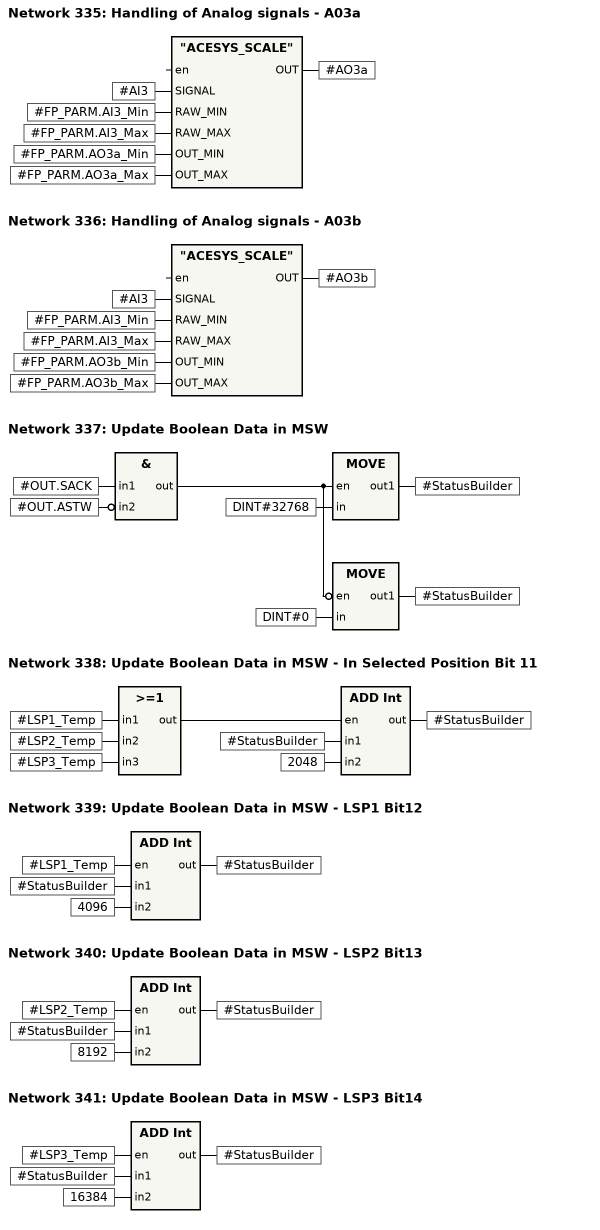
   "ACESYS_SCALE"(SIGNAL := #AI3,
                  RAW_MIN := #FP_PARM.AI3_Min,
                  RAW_MAX := #FP_PARM.AI3_Max,
                  OUT_MIN := #FP_PARM.AO3a_Min,
                  OUT_MAX := #FP_PARM.AO3a_Max,
                  OUT => #AO3a);
END_REGION

REGION Network 336: Handling of Analog signals - A03b
   "ACESYS_SCALE"(SIGNAL := #AI3,
                  RAW_MIN := #FP_PARM.AI3_Min,
                  RAW_MAX := #FP_PARM.AI3_Max,
                  OUT_MIN := #FP_PARM.AO3b_Min,
                  OUT_MAX := #FP_PARM.AO3b_Max,
                  OUT => #AO3b);
END_REGION

REGION Network 337: Update Boolean Data in MSW
   #_w1 := #OUT.SACK AND NOT #OUT.ASTW;
   IF #_w1 THEN #StatusBuilder := DINT#32768; END_IF;
   IF NOT #_w1 THEN #StatusBuilder := DINT#0; END_IF;
END_REGION

REGION Network 338: Update Boolean Data in MSW - In Selected Position Bit 11
   IF #LSP1_Temp OR #LSP2_Temp OR #LSP3_Temp THEN #StatusBuilder := #StatusBuilder + 2048; END_IF;
END_REGION

REGION Network 339: Update Boolean Data in MSW - LSP1 Bit12
   IF #LSP1_Temp THEN #StatusBuilder := #StatusBuilder + 4096; END_IF;
END_REGION

REGION Network 340: Update Boolean Data in MSW - LSP2 Bit13
   IF #LSP2_Temp THEN #StatusBuilder := #StatusBuilder + 8192; END_IF;
END_REGION

REGION Network 341: Update Boolean Data in MSW - LSP3 Bit14
   IF #LSP3_Temp THEN #StatusBuilder := #StatusBuilder + 16384; END_IF;
END_REGION

REGION Network 342: Update Boolean Data in MSW - Mode Info
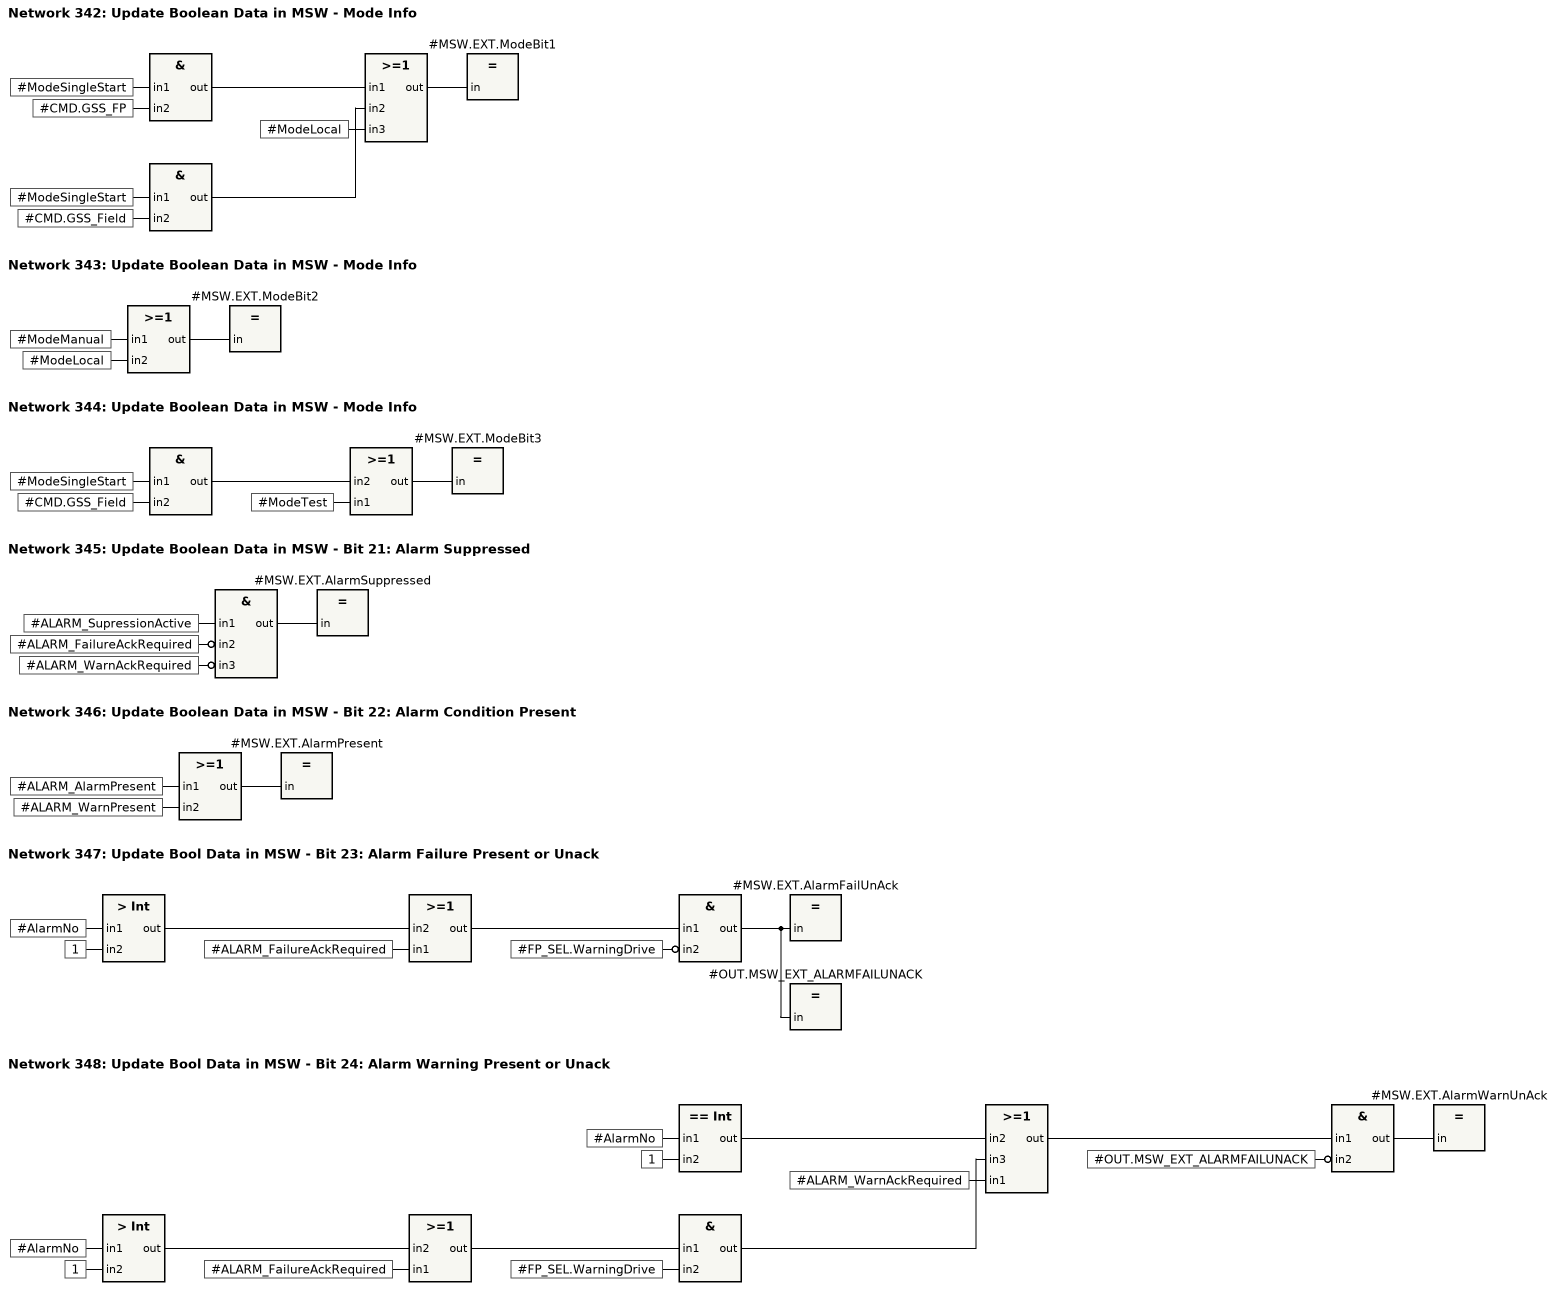
   #MSW.EXT.ModeBit1 := (#ModeSingleStart AND #CMD.GSS_FP) OR (#ModeSingleStart AND #CMD.GSS_Field) OR #ModeLocal;
END_REGION

REGION Network 343: Update Boolean Data in MSW - Mode Info
   #MSW.EXT.ModeBit2 := #ModeManual OR #ModeLocal;
END_REGION

REGION Network 344: Update Boolean Data in MSW - Mode Info
   #MSW.EXT.ModeBit3 := (#ModeSingleStart AND #CMD.GSS_Field) OR #ModeTest;
END_REGION

REGION Network 345: Update Boolean Data in MSW - Bit 21: Alarm Suppressed
   #MSW.EXT.AlarmSuppressed := #ALARM_SupressionActive AND NOT #ALARM_FailureAckRequired AND NOT #ALARM_WarnAckRequired;
END_REGION

REGION Network 346: Update Boolean Data in MSW - Bit 22: Alarm Condition Present
   #MSW.EXT.AlarmPresent := #ALARM_AlarmPresent OR #ALARM_WarnPresent;
END_REGION

REGION Network 347: Update Bool Data in MSW - Bit 23: Alarm Failure Present or Unack
   #MSW.EXT.AlarmFailUnAck := ((#AlarmNo > 1) OR #ALARM_FailureAckRequired) AND NOT #FP_SEL.WarningDrive;
   #OUT.MSW_EXT_ALARMFAILUNACK := #MSW.EXT.AlarmFailUnAck;
END_REGION

REGION Network 348: Update Bool Data in MSW - Bit 24: Alarm Warning Present or Unack
   #MSW.EXT.AlarmWarnUnAck := ((#AlarmNo = 1) OR (((#AlarmNo > 1) OR #ALARM_FailureAckRequired) AND #FP_SEL.WarningDrive) OR #ALARM_WarnAckRequired) AND NOT #OUT.MSW_EXT_ALARMFAILUNACK;
END_REGION

REGION Network 349: Update Boolean Data in MSW - Bit 25: Acknowledge Required
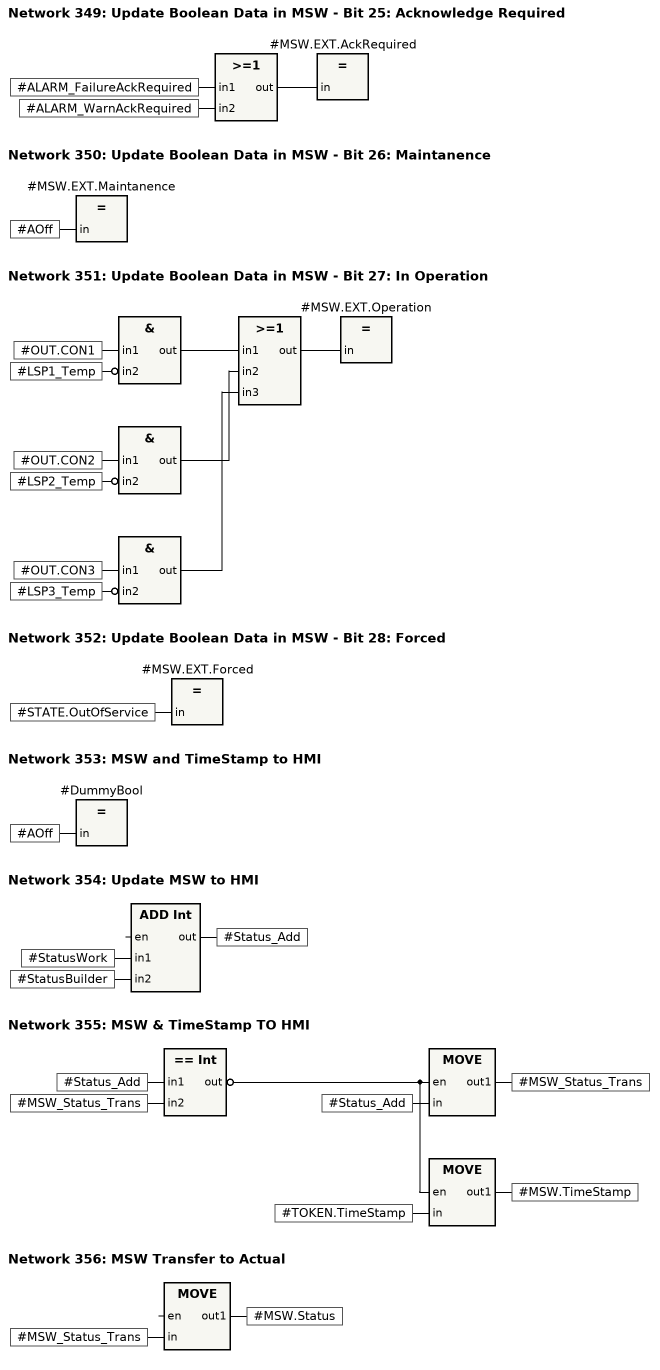
   #MSW.EXT.AckRequired := #ALARM_FailureAckRequired OR #ALARM_WarnAckRequired;
END_REGION

REGION Network 350: Update Boolean Data in MSW - Bit 26: Maintanence
   #MSW.EXT.Maintanence := #AOff;
END_REGION

REGION Network 351: Update Boolean Data in MSW - Bit 27: In Operation
   #MSW.EXT.Operation := (#OUT.CON1 AND NOT #LSP1_Temp) OR (#OUT.CON2 AND NOT #LSP2_Temp) OR (#OUT.CON3 AND NOT #LSP3_Temp);
END_REGION

REGION Network 352: Update Boolean Data in MSW - Bit 28: Forced
   // Build 002 - 27 March 2019 : State.OutOfService flag will set MSW.Ext.28 bit to enable force icon in Symbols
   #MSW.EXT.Forced := #STATE.OutOfService;
END_REGION

REGION Network 353: MSW and TimeStamp to HMI
   Done:
   #DummyBool := #AOff;
END_REGION

REGION Network 354: Update MSW to HMI
   #Status_Add := #StatusWork + #StatusBuilder;
END_REGION

REGION Network 355: MSW & TimeStamp TO HMI
   #_w1 := NOT (#Status_Add = #MSW_Status_Trans);
   IF #_w1 THEN
       #MSW_Status_Trans := #Status_Add;
       #MSW.TimeStamp := #TOKEN.TimeStamp;
   END_IF;
END_REGION

REGION Network 356: MSW Transfer to Actual
   #MSW.Status := #MSW_Status_Trans;
END_REGION

REGION Network 357: Update Token Data - Unit Alarm
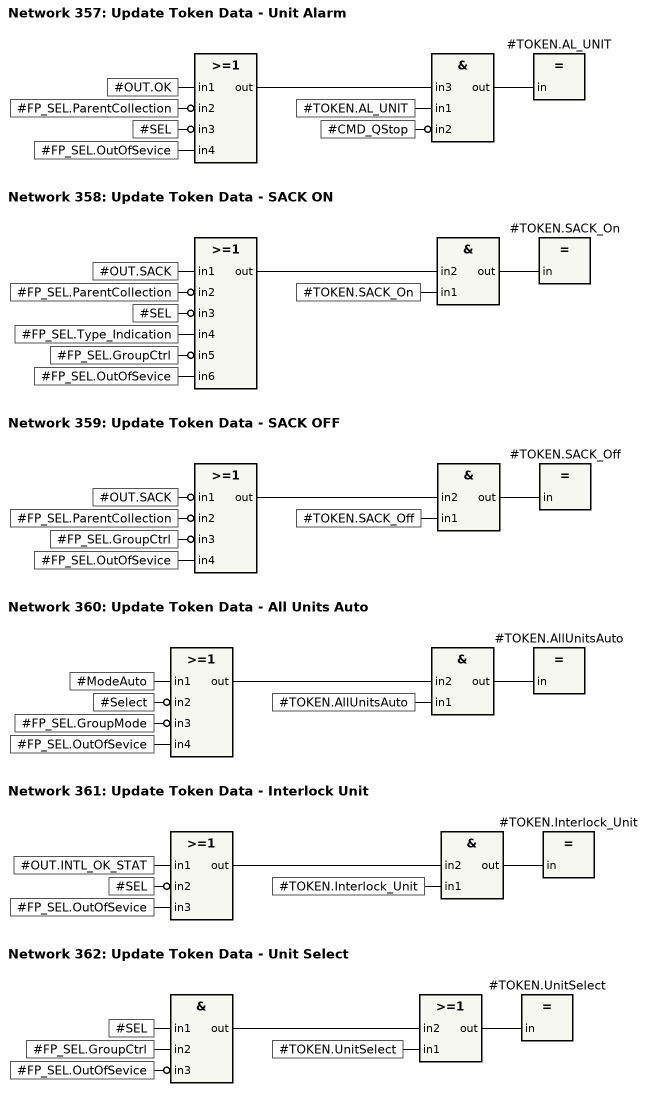
   #TOKEN.AL_UNIT := (#OUT.OK OR NOT #FP_SEL.ParentCollection OR NOT #SEL OR #FP_SEL.OutOfSevice) AND #TOKEN.AL_UNIT AND NOT #CMD_QStop;
END_REGION

REGION Network 358: Update Token Data - SACK ON
   // Build 006 - 24.Jun.2020 (MIA-US): Replace "Select" with "SEL" and "FP_SEL.Type_Indication"
   #TOKEN.SACK_On := (#OUT.SACK OR NOT #FP_SEL.ParentCollection OR NOT #SEL OR #FP_SEL.Type_Indication OR NOT #FP_SEL.GroupCtrl OR #FP_SEL.OutOfSevice) AND #TOKEN.SACK_On;
END_REGION

REGION Network 359: Update Token Data - SACK OFF
   #TOKEN.SACK_Off := (NOT #OUT.SACK OR NOT #FP_SEL.ParentCollection OR NOT #FP_SEL.GroupCtrl OR #FP_SEL.OutOfSevice) AND #TOKEN.SACK_Off;
END_REGION

REGION Network 360: Update Token Data - All Units Auto
   #TOKEN.AllUnitsAuto := (#ModeAuto OR NOT #Select OR NOT #FP_SEL.GroupMode OR #FP_SEL.OutOfSevice) AND #TOKEN.AllUnitsAuto;
END_REGION

REGION Network 361: Update Token Data - Interlock Unit
   #TOKEN.Interlock_Unit := (#OUT.INTL_OK_STAT OR NOT #SEL OR #FP_SEL.OutOfSevice) AND #TOKEN.Interlock_Unit;
END_REGION

REGION Network 362: Update Token Data - Unit Select
   #TOKEN.UnitSelect := (#SEL AND #FP_SEL.GroupCtrl AND NOT #FP_SEL.OutOfSevice) OR #TOKEN.UnitSelect;
END_REGION

REGION Network 363: Update Token Data - Start Warning
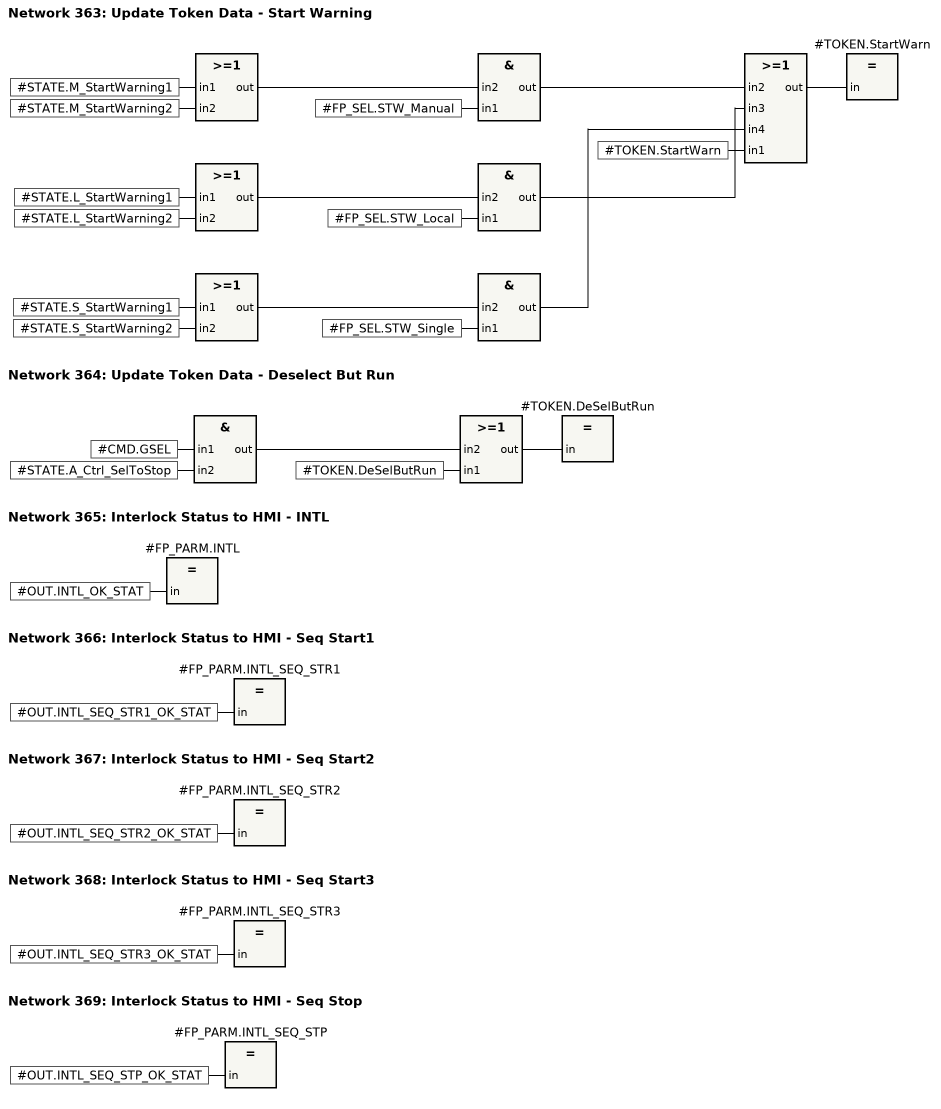
   #TOKEN.StartWarn := ((#STATE.M_StartWarning1 OR #STATE.M_StartWarning2) AND #FP_SEL.STW_Manual) OR ((#STATE.L_StartWarning1 OR #STATE.L_StartWarning2) AND #FP_SEL.STW_Local) OR ((#STATE.S_StartWarning1 OR #STATE.S_StartWarning2) AND #FP_SEL.STW_Single) OR #TOKEN.StartWarn;
END_REGION

REGION Network 364: Update Token Data - Deselect But Run
   #TOKEN.DeSelButRun := (#CMD.GSEL AND #STATE.A_Ctrl_SelToStop) OR #TOKEN.DeSelButRun;
END_REGION

REGION Network 365: Interlock Status to HMI - INTL
   #FP_PARM.INTL := #OUT.INTL_OK_STAT;
END_REGION

REGION Network 366: Interlock Status to HMI - Seq Start1
   #FP_PARM.INTL_SEQ_STR1 := #OUT.INTL_SEQ_STR1_OK_STAT;
END_REGION

REGION Network 367: Interlock Status to HMI - Seq Start2
   #FP_PARM.INTL_SEQ_STR2 := #OUT.INTL_SEQ_STR2_OK_STAT;
END_REGION

REGION Network 368: Interlock Status to HMI - Seq Start3
   #FP_PARM.INTL_SEQ_STR3 := #OUT.INTL_SEQ_STR3_OK_STAT;
END_REGION

REGION Network 369: Interlock Status to HMI - Seq Stop
   #FP_PARM.INTL_SEQ_STP := #OUT.INTL_SEQ_STP_OK_STAT;
END_REGION

REGION Network 370: Interlock Link
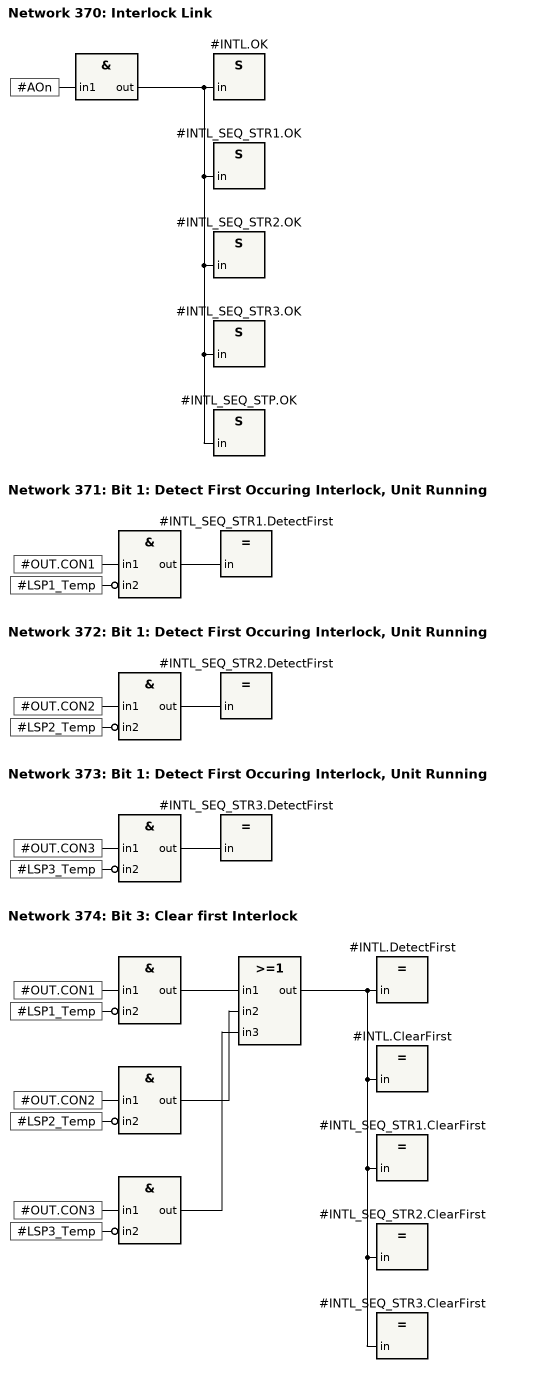
   IF #AOn THEN
       #INTL.OK := TRUE;
       #INTL_SEQ_STR1.OK := TRUE;
       #INTL_SEQ_STR2.OK := TRUE;
       #INTL_SEQ_STR3.OK := TRUE;
       #INTL_SEQ_STP.OK := TRUE;
   END_IF;
END_REGION

REGION Network 371: Bit 1: Detect First Occuring Interlock, Unit Running
   #INTL_SEQ_STR1.DetectFirst := #OUT.CON1 AND NOT #LSP1_Temp;
END_REGION

REGION Network 372: Bit 1: Detect First Occuring Interlock, Unit Running
   #INTL_SEQ_STR2.DetectFirst := #OUT.CON2 AND NOT #LSP2_Temp;
END_REGION

REGION Network 373: Bit 1: Detect First Occuring Interlock, Unit Running
   #INTL_SEQ_STR3.DetectFirst := #OUT.CON3 AND NOT #LSP3_Temp;
END_REGION

REGION Network 374: Bit 3: Clear first Interlock
   #INTL.DetectFirst := (#OUT.CON1 AND NOT #LSP1_Temp) OR (#OUT.CON2 AND NOT #LSP2_Temp) OR (#OUT.CON3 AND NOT #LSP3_Temp);
   #INTL.ClearFirst := #INTL.DetectFirst;
   #INTL_SEQ_STR1.ClearFirst := #INTL.DetectFirst;
   #INTL_SEQ_STR2.ClearFirst := #INTL.DetectFirst;
   #INTL_SEQ_STR3.ClearFirst := #INTL.DetectFirst;
END_REGION

REGION Network 375: Device Simulation - Sim Enable
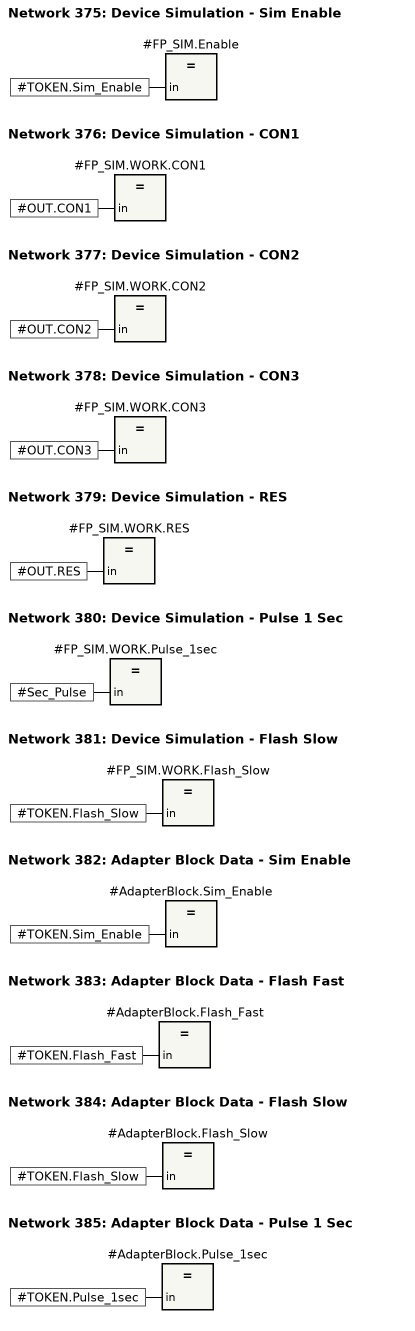
   #FP_SIM.Enable := #TOKEN.Sim_Enable;
END_REGION

REGION Network 376: Device Simulation - CON1
   #FP_SIM.WORK.CON1 := #OUT.CON1;
END_REGION

REGION Network 377: Device Simulation - CON2
   #FP_SIM.WORK.CON2 := #OUT.CON2;
END_REGION

REGION Network 378: Device Simulation - CON3
   #FP_SIM.WORK.CON3 := #OUT.CON3;
END_REGION

REGION Network 379: Device Simulation - RES
   #FP_SIM.WORK.RES := #OUT.RES;
END_REGION

REGION Network 380: Device Simulation - Pulse 1 Sec
   #FP_SIM.WORK.Pulse_1sec := #Sec_Pulse;
END_REGION

REGION Network 381: Device Simulation - Flash Slow
   #FP_SIM.WORK.Flash_Slow := #TOKEN.Flash_Slow;
END_REGION

REGION Network 382: Adapter Block Data - Sim Enable
   #AdapterBlock.Sim_Enable := #TOKEN.Sim_Enable;
END_REGION

REGION Network 383: Adapter Block Data - Flash Fast
   #AdapterBlock.Flash_Fast := #TOKEN.Flash_Fast;
END_REGION

REGION Network 384: Adapter Block Data - Flash Slow
   #AdapterBlock.Flash_Slow := #TOKEN.Flash_Slow;
END_REGION

REGION Network 385: Adapter Block Data - Pulse 1 Sec
   #AdapterBlock.Pulse_1sec := #TOKEN.Pulse_1sec;
END_REGION

REGION Network 386: Adapter Block Data - LOC
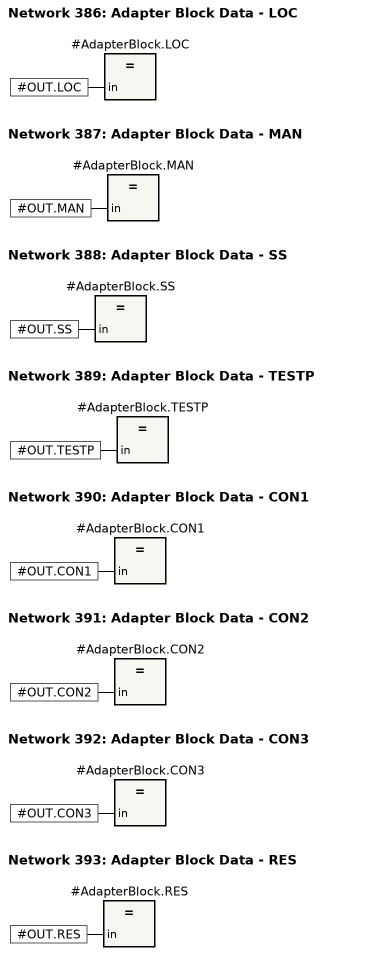
   #AdapterBlock.LOC := #OUT.LOC;
END_REGION

REGION Network 387: Adapter Block Data - MAN
   #AdapterBlock.MAN := #OUT.MAN;
END_REGION

REGION Network 388: Adapter Block Data - SS
   #AdapterBlock.SS := #OUT.SS;
END_REGION

REGION Network 389: Adapter Block Data - TESTP
   #AdapterBlock.TESTP := #OUT.TESTP;
END_REGION

REGION Network 390: Adapter Block Data - CON1
   #AdapterBlock.CON1 := #OUT.CON1;
END_REGION

REGION Network 391: Adapter Block Data - CON2
   #AdapterBlock.CON2 := #OUT.CON2;
END_REGION

REGION Network 392: Adapter Block Data - CON3
   #AdapterBlock.CON3 := #OUT.CON3;
END_REGION

REGION Network 393: Adapter Block Data - RES
   #AdapterBlock.RES := #OUT.RES;
END_REGION

REGION Network 394: Write STAT to OUT
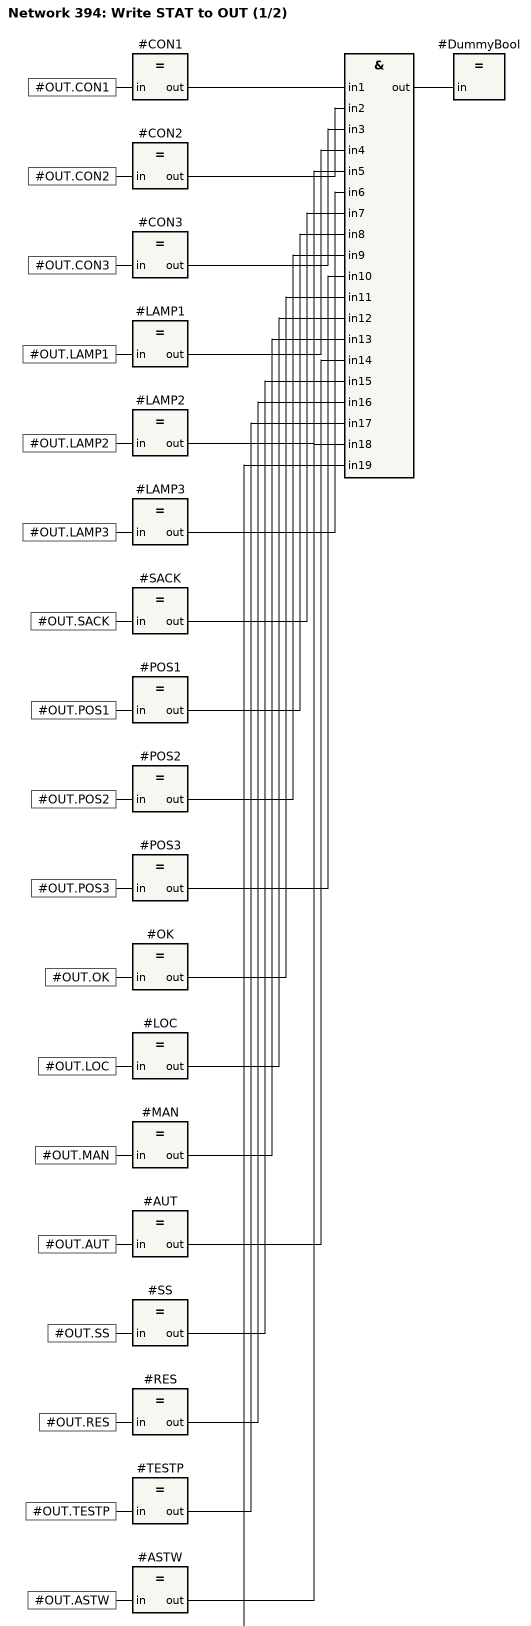
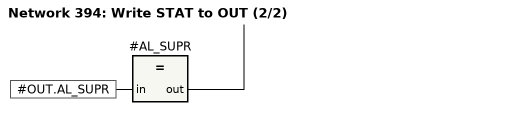
   #CON1 := #OUT.CON1;
   #CON2 := #OUT.CON2;
   #CON3 := #OUT.CON3;
   #LAMP1 := #OUT.LAMP1;
   #LAMP2 := #OUT.LAMP2;
   #LAMP3 := #OUT.LAMP3;
   #SACK := #OUT.SACK;
   #POS1 := #OUT.POS1;
   #POS2 := #OUT.POS2;
   #POS3 := #OUT.POS3;
   #OK := #OUT.OK;
   #LOC := #OUT.LOC;
   #MAN := #OUT.MAN;
   #AUT := #OUT.AUT;
   #SS := #OUT.SS;
   #RES := #OUT.RES;
   #TESTP := #OUT.TESTP;
   #ASTW := #OUT.ASTW;
   #AL_SUPR := #OUT.AL_SUPR;
   #DummyBool := #OUT.CON1 AND #OUT.CON2 AND #OUT.CON3 AND #OUT.LAMP1 AND #OUT.LAMP2 AND #OUT.LAMP3 AND #OUT.SACK AND #OUT.POS1 AND #OUT.POS2 AND #OUT.POS3 AND #OUT.OK AND #OUT.LOC AND #OUT.MAN AND #OUT.AUT AND #OUT.SS AND #OUT.RES AND #OUT.TESTP AND #OUT.ASTW AND #OUT.AL_SUPR;
END_REGION
END_FUNCTION_BLOCK

FUNCTION_BLOCK "ACESYS_SCHENCK"   // FB215, FBD
TITLE = ACESYS V8.0 - Build 006 - SCHENCK FEEDER
{ S7_Optimized_Access := 'FALSE' }
AUTHOR : FLSmidth
FAMILY : ACESYS
NAME : SCHENCK
VERSION : 8.0
   VAR_INPUT
      CMD : "ACESYS_GRP_CMD";
      INREF : Int;   // Address reference for Input data
      OUTREF : Int;   // Address reference for Output data
      NET : Int;   // Net number
      NODE : Int;   // Node Number
      FUNCTYPE : Int;   // Function Type (1= Disocont / 2= Intecont)
      OPTIONS : Int;   // Operation Options
      SEL : Bool := TRUE;   // Unit Select by User program
      ASTR : Bool := TRUE;   // Auto Start
      SSW : Bool := TRUE;   // Service switch
      FSTOP : Bool;   // Filling Devices stopped
      SP : Real;   // Set Point
   END_VAR
   VAR_OUTPUT
      INTL : "ACESYS_INTL";   // Interlock
      INTL_SEQ_STR : "ACESYS_INTL";   // Interlock Sequence Start
      INTL_SEQ_STP : "ACESYS_INTL";   // Interlock Sequence Stop
      LAMP : Bool;   // Lamp 1
      SACK : Bool;   // Start Acknowledge
      RD : Bool;   // Run delayed 1
      RUN : Bool;   // Run 1
      OK : Bool;   // Unit Status OK (no alarms)
      LOC : Bool;   // Unit in Local Mode
      MAN : Bool;   // Unit in Manual Mode
      AUT : Bool;   // Unit in Auto Mode
      SS : Bool;   // Unit in Single Start Mode
      TESTP : Bool;   // Test mode permission to unit
      ASTW : Bool;   // Start warning
      AL_SUPR : Bool;   // Supress Child Alarms
      WCSEL : Bool;   // Weight Check Selected
      WCRUN : Bool;   // Weight Check Active
      WCFIN : Bool;   // Weight Check Finished
      FILL_BIN : Bool;   // Start Silo feeding system
      CORR_Factor : Real;   // Acutal Correction [Factor]
      CORR_Pct : Real;   // Acutal Coorrection [%]
      FEED_Pct : Real;   // Actual Feed [&]
      FEED_Eng : Real;   // Actual Feed [t/h]
      WEIGHT_Pct : Real;   // Actual Bin Weight [%]
      WEIGHT_Eng : Real;   // Actual Bin Weight [t]
      WSP_Pct : Real;   // Actual Working Setpoint [%]
      WSP_Eng : Real;   // Actual Working Setpoint [t/h]
      SP_Pct : Real;   // Setpoint to Feeder [%]
      SP_Eng : Real;   // Setpoint to Feeder [t/h]
      TOTAL : Real;   // Totalizer (t)
      MSW : "ACESYS_HMI_STAT_32T";
   END_VAR
   VAR_IN_OUT
      TOKEN : "ACESYS_TOKEN";
   END_VAR
   VAR
      BlockInfo : Struct
         Ace_Version : Int;   // Acesys Block Version Number
         Ace_BuildNo : Int;   // Acesys Block Build Number
         State_Act : Int;   // Actual State Number
         State_Prev : Int;   // Previous State Number
         DB_Number : Int;   // Block Instance DB Number
      END_STRUCT;
      FP_CMD : Struct   // Faceplate Commands
         QuickStop : Bool;
         StartCalibration : Bool;
         AcceptCalcResult : Bool;
         AbortCalibration : Bool;
         ResetTotalizer : Bool;
         Spare_13 : Bool;
         Spare_14 : Bool;
         AckAlarm : Bool;
         Auto : Bool;
         Manual : Bool;
         Local : Bool;
         Start : Bool;
         Spare1 : Bool;
         Stop : Bool;
         Reset : Bool;
         Test : Bool;
      END_STRUCT;
      FP_SEL : Struct   // Faceplate Selections
         STW_AutoStart : Bool;   // Faceplate Start Warning in Auto Start mode
         STW_Manual : Bool;   // Faceplate Start Warning in Manual mode
         STW_Single : Bool;   // Faceplate Start Warning in Single Start mode
         Spare8 : Bool;
         ParentSupress : Bool;   // Enable Parent Supress of alarms
         ParentCollection : Bool;   // Enable Inching in Manual Mode
         INCH_Man : Bool;   // Enable Inching in Manual Mode
         OutOfSevice : Bool;   // Select Out of Service
         Spare3 : Bool;
         WarningDrive : Bool;   // 0 = Failure Drive / 1 = Warning Drive
         Volumetric : Bool;
         Gravametric : Bool;
         Spare5 : Bool;
         Spare4 : Bool;
         Spare2 : Bool;
         Spare1 : Bool;
      END_STRUCT;
      FP_EN : Struct
         Mode_Auto : Bool;
         Mode_Man : Bool;
         Mode_Loc : Bool;
         Mode_Test : Bool;
         Mode_SS_Field : Bool;
         Mode_SS_FP : Bool;
         PB_QStop : Bool;
         Spare9 : Bool;
         Spare8 : Bool;
         Spare7 : Bool;
         Spare6 : Bool;
         Spare5 : Bool;
         Spare4 : Bool;
         Spare3 : Bool;
         Spare2 : Bool;
         Spare1 : Bool;
      END_STRUCT;
      FP_DIM : Struct   // Faceplate Dimmed Buttons
         Auto : Bool;
         Local : Bool;
         Manual : Bool;
         Start : Bool;
         Stop : Bool;
         Test : Bool;
         QStop : Bool;
         StartCalibration : Bool;
         AcceptCalcResult : Bool;
         AbortCalibration : Bool;
         ResetTotalizer : Bool;
         Spare3 : Bool;
         Spare2 : Bool;
         Spare1 : Bool;
      END_STRUCT;
      FP_PARM : Struct   // Faceplate Parameters
         StartWarn_Pre : Int;
         StartWarn_Acc : Int;
         RunDelay_Pre : Int;
         RunDelay_Acc : Int;
         DelayStart_Pre : Int;
         DelayStart_Acc : Int;
         DelayStop_Pre : Int;
         DelayStop_Acc : Int;
         ReturnMon_Pre : Int;
         ReturnMon_Acc : Int;
         StopReason : Int;
         UserParameter : Int;   // Selectable parameter to be read from Schenck
         FEED_max : Real := 100.0;   // Actual Feed max
         FEED_min : Real;   // Actual Feed min
         WEIGHT_max : Real := 100.0;   // Actual Bin Weight max
         WEIGHT_min : Real;   // Actual Bin Weight min
         EventCode : Int;   // Schenck event code to ECS (No. + Group)
         EventNo : Byte;   // Schenck event number to ECS
         EventGrp : Byte;   // Schenck event group to ECS
         EventClass : Byte;   // Schenck event class to ECS
         EventAck : Byte;   // Schenck event acknowledge status to ECS
         INTL : Bool;   // Interlock
         INTL_SEQ_STR : Bool;   // Interlock Sequence Start
         INTL_SEQ_STP : Bool;   // Interlock Sequence Stop
         Spare13 : Bool;
         Spare12 : Bool;
         Spare11 : Bool;
         Spare10 : Bool;
         Spare09 : Bool;
         Spare08 : Bool;
         Spare07 : Bool;
         Spare06 : Bool;
         Spare05 : Bool;
         Spare04 : Bool;
         Spare03 : Bool;
         Spare02 : Bool;
         Spare01 : Bool;
      END_STRUCT;
      Rx : Struct
         SB00_0_NormMode : Bool;   // Normal Mode
         SB00_1_KBMode : Bool;   // Keyboard Mode
         SB00_2_LocMode : Bool;   // Local Mode
         SB00_3_SimMode : Bool;   // Simulation Mode
         SB00_4 : Bool;   // Volum. Start-Up
         SB00_5 : Bool;   // Meas. Drive On
         SB00_6 : Bool;   // Wheel Meas. Drive Delay
         SB00_7 : Bool;   // Setpoint Limited
         SB01_0_ScaleOn : Bool;   // Scale On (RET)
         SB01_1_NotRel : Bool;   // Not Released
         SB01_2 : Bool;   // Counter Active
         SB01_3_VolMode : Bool;   // Volumetric Mode
         SB01_4 : Bool;   // Select Langugage Ok
         SB01_5_Alarm : Bool;   // Alarm
         SB01_6_Warn : Bool;   // Warning
         SB01_7_CalActive : Bool;   // Calibration Active
         SB02_0 : Bool;   // Tare
         SB02_1 : Bool;   // Zero Set
         SB02_2 : Bool;   // Weight Check
         SB02_3 : Bool;   // Pulses/Revolution
         SB02_4 : Bool;   // DAE Adjustment
         SB02_5 : Bool;   // Auto Zero Active
         SB02_6 : Bool;   // Volumetric Adaption
         SB02_7 : Bool;   // Gravimetric Optimization
         SB03_0 : Bool;   // Batch Selected
         SB03_1 : Bool;   // Batch Active
         SB03_2 : Bool;   // Batch Dribble Feed (Pre-act Cont.)
         SB03_3 : Bool;   // Batch + Clearance
         SB03_4 : Bool;   // NON-SI Active
         SB03_5 : Bool;   // Dead Time Active
         SB03_6 : Bool;   // Dead Time Setpoint Active
         SB03_7 : Bool;   // Dead Time ON/OFF Active
         SD04_FeedRate : Real;   // Feed Rate [kg/h]
         SD08_Totalizer1 : Real;   // Totalizer 1 [kg]
         SD12_BinWeight : Real;   // Bin Weigher Fill Weight [kg]
         SB16_SoftRev : Byte;   // Software Revision
         SB17_ScaleType : Byte;   // Scale Type
         SW18_SoftVer : Word;   // Software Version
         SB20_0 : Bool;   // KME Active
         SB20_1 : Bool;   // No Alarm
         SB20_2 : Bool;   // No Warning
         SB20_3 : Bool;   // Pulse counter reading
         SB20_4_NoDev : Bool;   // No Deviation
         SB20_5_Ready : Bool;   // Ready
         SB20_6 : Bool;   // KME Rel Tare Not Exceeded
         SB20_7 : Bool;   // KME Abs. Tare Not Exceeded
         SB21_0 : Bool;   // Calibr. Set Norminal Feed Rate
         SB21_1 : Bool;   // Pre-cut-off amount Dig. Output
         SB21_2 : Bool;   // MAX Limit Value
         SB21_3 : Bool;   // MIN Limit Value
         SB21_4 : Bool;   // VSM 20110 (DISOCONT L)
         SB21_5 : Bool;   // Make-up active
         SB21_6 : Bool;   // VSM 20107 (pulverized coal)
         SB21_7_FillBin : Bool;   // Fill Bin Weigher
         SB22 : Byte;   // Standby
         SB23_0 : Bool;   // KME Rel. Range Not Exceeded
         SB23_1 : Bool;   // KME Abs. Range Not Exceeded
         SB23_2 : Bool;   // VSM Type A (big)
         SB23_3 : Bool;   // VSM Type F (fast)
         SB23_4 : Bool;
         SB23_5 : Bool;
         SB23_6 : Bool;
         SB23_7 : Bool;
         SB24_EventHI : Byte;   // Highest-Priority Event (HI)
         SB25_EventLO : Byte;   // Highest-Priority Event (LO)
         SB26 : Byte;   // Number in parameter block
         SB27 : Byte;   // Parameter block including the event class
         SD28 : Real;   // User selected parameter from faceplate
         SB32_0 : Bool;   // Feed Rate > Max
         SB32_1 : Bool;   // Feed Rate < Min
         SB32_2 : Bool;   // Belt Load > Max
         SB32_3 : Bool;   // Belt Load < Min
         SB32_4 : Bool;   // Speed > Max
         SB32_5 : Bool;   // Speed < Min
         SB32_6 : Bool;   // Bin > Max
         SB32_7 : Bool;   // Bin < Min
         SB33_0 : Bool;   // Meas. System
         SB33_1 : Bool;   // Gain-In-Weight
         SB33_2 : Bool;   // Filling Active
         SB33_3_Discharge : Bool;   // Discharge Active
         SB33_4 : Bool;   // Gate Open
         SB33_5 : Bool;   // Gate Closed
         SB33_6 : Bool;   // 2nd Batch Unit Active (VLW20151 only)
         SB33_7_Hopper : Bool;   // Surge Hopper present
         SB34_0_CheckAvail : Bool;   // 8 - Check System Available
         SB34_1_RelTaraExc : Bool;   // Rel. tare Exceeded
         SB34_2_AbsTaraExc : Bool;   // Abs. tare Exceeded
         SB34_3_RelRangeExc : Bool;   // Rel. range Exceeded
         SB34_4_AbsRangeExc : Bool;   // Abs. range Exceeded
         SB34_5 : Bool;   // Check Meas. Announced
         SB34_6_Prepare : Bool;   // Prepare Check
         SB34_7_CheckActive : Bool;   // Check Active
         SB35_0 : Bool;   // Bin Level Control existent
         SB35_1 : Bool;   // Hopper level > Max
         SB35_2 : Bool;   // Hopper level < Min
         SB35_3 : Bool;   // Measured load > Max
         SB35_4 : Bool;   // Measured load < Min
         SB35_5 : Bool;   // n > Max
         SB35_6 : Bool;   // n < Min
         SB35_7_CheckWaitAck : Bool;   // Check System waits for acknowledgement
         SD36_CheckResult : Real;   // Check Result F/Z [Factor] 1=0%
         SD40_ActSP : Real;   // Actual Setpoint [kg/h]
         SD44_Deviation : Real;   // Deviation
         SD48 : Real;   // Not Used
         SD52 : Real;   // Not Used
      END_STRUCT;
      Tx : Struct
         CB02_0 : Bool;   // Command 4 (HI): Volm. Synchronous
         CB02_1 : Bool;   // Command 4 (HI): Moisture Corr. On
         CB02_2 : Bool;   // Command 4 (HI): Moisture Corr. Off
         CB02_3 : Bool;   // Command 4 (HI): Meas. Drive Off
         CB02_4 : Bool;   // Command 4 (HI): Gate Feedback
         CB02_5 : Bool;   // Command 4 (HI): Open Gate Manual
         CB02_6 : Bool;   // Command 4 (HI): Stop Gate Manual
         CB02_7 : Bool;   // Command 4 (HI): Close Gate Manual
         CB03_0_StrScale : Bool;   // Command 4 (LO): Start Scale
         CB03_1_StpScale : Bool;   // Command 4 (LO): Stop Scale
         CB03_2_ClearEvent : Bool;   // Command 4 (LO): Clear Events (RESET)
         CB03_3_Release : Bool;   // Command 4 (LO): Release
         CB03_4_SelVol : Bool;   // Command 4 (LO): Select Volumetrice Mode
         CB03_5_SelGrav : Bool;   // Command 4 (LO): Select Gravimetric Mode
         CB03_6_ResTot : Bool;   // Command 4 (LO): Reset Totalizer 1
         CB03_7 : Bool;   // Command 4 (LO): Reset Totalizer 2
         CB04_0 : Bool;   // Command 5 (HI): Filling Start
         CB04_1 : Bool;   // Command 5 (HI): Filling Stop
         CB04_2 : Bool;   // Command 5 (HI): Emptying Start
         CB04_3 : Bool;   // Command 5 (HI): Emptying Stop
         CB04_4 : Bool;   // Command 5 (HI): Init .Hopper Controller
         CB04_5 : Bool;   // Command 5 (HI): Activate Fill Unit
         CB04_6 : Bool;   // Command 5 (HI): Activate Prefeeder
         CB04_7 : Bool;   // Command 5 (HI): Stop Prefeeder
         CB05_0 : Bool;   // Command 5 (LO): Select Batch
         CB05_1 : Bool;   // Command 5 (LO): Deselect Batch
         CB05_2 : Bool;   // Command 5 (LO): Abort Batch
         CB05_3 : Bool;   // Command 5 (LO): Next Batch + Clearance
         CB05_4 : Bool;   // Command 5 (LO): Make-Up
         CB05_5 : Bool;   // Command 5 (LO): Emergency Setpoint On
         CB05_6 : Bool;   // Command 5 (LO): Emergency Setpoint Off
         CB05_7 : Bool;   // Command 5 (LO): Meas Drive On
         CB14_0 : Bool;   // Command 6 (HI): Bin controller Autom.
         CB14_1 : Bool;   // Command 6 (HI): Bin controller Manual
         CB14_2 : Bool;   // Command 6 (HI): Bin controller Man. Start
         CB14_3 : Bool;   // Command 6 (HI): Bin controller Man Stop
         CB14_4 : Bool;   // Command 6 (HI): Optimization Bin Controller
         CB14_5 : Bool;   // Command 6 (HI): Print check Meas. Result
         CB14_6 : Bool;   // Command 6 (HI): Dead Time preassign
         CB14_7 : Bool;   // Command 6 (HI): Dead Time initialize
         CB15_0_StrTara : Bool;   // Command 6 (LO): Start internal check for tara
         CB15_1_StrRange : Bool;   // Command 6 (LO): Start internal check for range
         CB15_2_Acquire : Bool;   // Command 6 (LO): Acquire check result
         CB15_3_Cancel : Bool;   // Command 6 (LO): Cancel check measurement
         CB15_4 : Bool;   // Command 6 (LO): Release check system
         CB15_5 : Bool;   // Command 6 (LO): Acquire ext. corr. factor for tare
         CB15_6 : Bool;   // Command 6 (LO): Acquire ext. corr. factor for range
         CB15_7 : Bool;   // Command 6 (LO): Start external check
         CB16_0 : Bool;   // Command 7 (HI): Linearization P4
         CB16_1 : Bool;   // Command 7 (HI): Volmetric
         CB16_2 : Bool;   // Command 7 (HI): Optimize controller
         CB16_3 : Bool;   // Command 7 (HI): Calibration Acquire
         CB16_4 : Bool;   // Command 7 (HI): Calibration Abort
         CB16_5 : Bool;   // Command 7 (HI): Time Acquire
         CB16_6 : Bool;   // Command 7 (HI): Bin: Tare
         CB16_7 : Bool;   // Command 7 (HI): Bin: Weight Check
         CB17_0 : Bool;   // Command 7 (LO): Tare
         CB17_1 : Bool;   // Command 7 (LO): Zero Set
         CB17_2 : Bool;   // Command 7 (LO): Weight Check
         CB17_3 : Bool;   // Command 7 (LO): Pulses/Revolution
         CB17_4 : Bool;   // Command 7 (LO): DAE Adjustment
         CB17_5 : Bool;   // Command 7 (LO): Liniarization P1
         CB17_6 : Bool;   // Command 7 (LO): Liniarization P2
         CB17_7 : Bool;   // Command 7 (LO): Liniarization P3
         CB20_0 : Bool;   // Command 10 (HI): Reset Sum of Component 9
         CB20_1 : Bool;   // Command 10 (HI): Reset Sum of Component 10
         CB20_2 : Bool;   // Command 10 (HI): Reset Sum of Batches
         CB20_3_FillStopped : Bool;   // Command 10 (HI): Filling Stopped
         CB20_4 : Bool;   // Command 10 (HI): Start (static)
         CB20_5 : Bool;   // Command 10 (HI):
         CB20_6 : Bool;   // Command 10 (HI): Activate 2nd Batch Unit
         CB20_7 : Bool;   // Command 10 (HI): De-activate 2nd Batch Unit
         CB21_0 : Bool;   // Command 10 (LO): Reset Sum of Component 1
         CB21_1 : Bool;   // Command 10 (LO): Reset Sum of Component 2
         CB21_2 : Bool;   // Command 10 (LO): Reset Sum of Component 3
         CB21_3 : Bool;   // Command 10 (LO): Reset Sum of Component 4
         CB21_4 : Bool;   // Command 10 (LO): Reset Sum of Component 5
         CB21_5 : Bool;   // Command 10 (LO): Reset Sum of Component 6
         CB21_6 : Bool;   // Command 10 (LO): Reset Sum of Component 7
         CB21_7 : Bool;   // Command 10 (LO): Reset Sum of Component 8
         CB22_0 : Bool;   // Command 11 (HI): Feeder 1 Active
         CB22_1 : Bool;   // Command 11 (HI): Feeder 1 Not Active
         CB22_2 : Bool;   // Command 11 (HI): Feeder 1 Active
         CB22_3 : Bool;   // Command 11 (HI): Feeder 1 Not Active
         CB22_4 : Bool;   // Command 11 (HI): Set Norminal Feed Rate
         CB22_5 : Bool;   // Command 11 (HI): Copy feed index block
         CB22_6 : Bool;   // Command 11 (HI):
         CB22_7 : Bool;   // Command 11 (HI):
         CB23 : Byte;   // Command 11 (LO): Component Number (1 Byte)
      END_STRUCT;
      FP_SHOW : Struct   // Faceplate Show Buttons
         PB_Auto : Bool;
         PB_Local : Bool;
         PB_Manual : Bool;
         PB_Start : Bool;
         PB_Stop : Bool;
         PB_Test : Bool;
         PB_QStop : Bool;
         SSW : Bool;
         Spare06 : Bool;
         ASTR : Bool;
         Spare07 : Bool;
         Spare05 : Bool;
         Spare04 : Bool;
         Spare03 : Bool;
         Spare02 : Bool;
         Spare01 : Bool;
      END_STRUCT;
      FP_SIM : "ACESYS_SIM_SCHENCK";
      STATE : Struct
         A_AutoStart : Bool;
         A_DelayedStart : Bool;
         A_DelayedStop : Bool;
         A_Running : Bool;
         A_Selected : Bool;
         A_SelToStop : Bool;
         A_Stopping : Bool;
         A_SeqStart : Bool;
         A_SeqStop : Bool;
         A_Starting : Bool;
         A_StartWarning : Bool;
         A_Stopped : Bool;
         S_AutoStart : Bool;
         S_Running : Bool;
         S_Starting : Bool;
         S_StartWarning : Bool;
         S_Stopped : Bool;
         M_Running : Bool;
         M_Starting : Bool;
         M_StartWarning : Bool;
         M_Stopped : Bool;
         L_Running : Bool;
         L_Stopped : Bool;
         T_TestMode : Bool;
         T_TestPermission : Bool;
         Alarm : Bool;
         Interlock : Bool;
         EmergencyStop : Bool;
         OutOfService : Bool;
      END_STRUCT;
      ONS : Struct
         AckAlarm : Bool;
         Cmd_Auto : Bool;
         Cmd_Manual : Bool;
         CMD_Local : Bool;
         CMD_Test : Bool;
         GLTP : Bool;
         RET : Bool;
         CMD_StartOff : Bool;
         CMD_StartON : Bool;
         SecPulse1 : Bool;
         SecPulse2 : Bool;
         Cal_Run : Bool;
         Cal_Sel : Bool;
         Cal_Start : Bool;
         Cal_Accept : Bool;
         Cal_Cancel : Bool;
         Volumetric : Bool;
         Gravametric : Bool;
         ResetTotalizer : Bool;
         Spare13 : Bool;
         Spare12 : Bool;
         Spare11 : Bool;
         Spare10 : Bool;
         Spare09 : Bool;
         Spare08 : Bool;
         Spare07 : Bool;
         Spare06 : Bool;
         Spare05 : Bool;
         Spare04 : Bool;
         Spare03 : Bool;
         Spare02 : Bool;
         Spare01 : Bool;
      END_STRUCT;
      StatusWork : Int;
      ModePointer : Int;
      AlarmNo : Int;
      AlarmNo_Old : Int;
      StartWarn_Mem : Int;
      RunDelay_Mem : Int;
      DelayStart_Mem : Int;
      DelayStop_Mem : Int;
      ReturnMon_Mem : Int;
      CMDDelay_Mem : Int;
      CalcAccept_Mem : Int;
      CalCancel_Mem : Int;
      ResetTot_Mem : Int;
      ModeAuto : Bool;
      ModeLocal : Bool;
      ModeManual : Bool;
      ModeSingleStart : Bool;
      ModeTest : Bool;
      Select : Bool;   // Parent & Program Select
      CMD_AckAlarm : Bool;
      CMD_Start : Bool;
      CMD_Stop : Bool;
      CMD_QStop : Bool;
      CMD_Reset : Bool;
      FromStateAuto : Bool;
      FromStateSingle : Bool;
      FromStateManual : Bool;
      FromStateLocal : Bool;
      FromStateTest : Bool;
      FromStopState : Bool;
      ALARM_SupressionActive : Bool;
      ALARM_AlarmPresent : Bool;
      ALARM_WarnPresent : Bool;
      ALARM_FailureAckRequired : Bool;
      ALARM_WarnAckRequired : Bool;
      StartWarn_TT : Bool;
      StartWarn_Done : Bool;
      Rundelay_Done : Bool;
      DelayStart_Done : Bool;
      DelayStop_Done : Bool;
      ReturnMon_Done : Bool;
      Trig_RET_ALARM : Bool;
      RET_OneScan : Bool;
      NotEmpty : Bool;   // Unit Stopped un-normal
      LSTR_Puls : Bool;
      Sec_Pulse : Bool;
      Reset : Bool;
      Cal_Start : Bool;
      Cal_Accept : Bool;
      Cal_Cancel : Bool;
      Cal_Accept_Time : Bool;
      Cal_Cancel_Time : Bool;
      Reset_Tot_Time : Bool;
      ResetTotalizer : Bool;
      OUT : Struct
         LAMP : Bool;
         SACK : Bool;
         RD : Bool;
         RUN : Bool;
         OK : Bool;
         LOC : Bool;
         MAN : Bool;
         AUT : Bool;
         SS : Bool;
         TESTP : Bool;
         ASTW : Bool;
         AL_SUPR : Bool;
         WCSEL : Bool;
         WCRUN : Bool;
         WCFIN : Bool;
         FILL_BIN : Bool;
         INTL_OK_STAT : Bool;
         INTL_SEQ_STR_OK_STAT : Bool;
         INTL_SEQ_STP_OK_STAT : Bool;
         MSW_EXT_ALARMFAILUNACK : Bool;
      END_STRUCT;
      MSW_Status_Trans : Int;
   END_VAR
   VAR_TEMP
      DISOCONT : Struct
         Tx_CW00 : Int;   // Command ID 1: Command 4+5 (140 Hex / 320 Dec)
         Tx_CB02_0 : Bool;   // Command 4 (HI): Volm. Synchronous
         Tx_CB02_1 : Bool;   // Command 4 (HI): Moisture Corr. On
         Tx_CB02_2 : Bool;   // Command 4 (HI): Moisture Corr. Off
         Tx_CB02_3 : Bool;   // Command 4 (HI): Meas. Drive Off
         Tx_CB02_4 : Bool;   // Command 4 (HI): Gate Feedback
         Tx_CB02_5 : Bool;   // Command 4 (HI): Open Gate Manual
         Tx_CB02_6 : Bool;   // Command 4 (HI): Stop Gate Manual
         Tx_CB02_7 : Bool;   // Command 4 (HI): Close Gate Manual
         Tx_CB03_0_StrScale : Bool;   // Command 4 (LO): Start Scale
         Tx_CB03_1_StpScale : Bool;   // Command 4 (LO): Stop Scale
         Tx_CB03_2_ClearEvent : Bool;   // Command 4 (LO): Clear Events (RESET)
         Tx_CB03_3_Release : Bool;   // Command 4 (LO): Release
         Tx_CB03_4_SelVol : Bool;   // Command 4 (LO): Select Volumetric Mode
         Tx_CB03_5_SelGrav : Bool;   // Command 4 (LO): Select Gravimetric Mode
         Tx_CB03_6_ResTot : Bool;   // Command 4 (LO): Reset Totalizer 1
         Tx_CB03_7 : Bool;   // Command 4 (LO): Reset Totalizer 2
         Tx_CB04_0 : Bool;   // Command 5 (HI): Filling Start
         Tx_CB04_1 : Bool;   // Command 5 (HI): Filling Stop
         Tx_CB04_2 : Bool;   // Command 5 (HI): Emptying Start
         Tx_CB04_3 : Bool;   // Command 5 (HI): Emptying Stop
         Tx_CB04_4 : Bool;   // Command 5 (HI): Init .Hopper Controller
         Tx_CB04_5 : Bool;   // Command 5 (HI): Activate Fill Unit
         Tx_CB04_6 : Bool;   // Command 5 (HI): Activate Prefeeder
         Tx_CB04_7 : Bool;   // Command 5 (HI): Stop Prefeeder
         Tx_CB05_0 : Bool;   // Command 5 (LO): Select Batch
         Tx_CB05_1 : Bool;   // Command 5 (LO): Deselect Batch
         Tx_CB05_2 : Bool;   // Command 5 (LO): Abort Batch
         Tx_CB05_3 : Bool;   // Command 5 (LO): Next Batch + Clearance
         Tx_CB05_4 : Bool;   // Command 5 (LO): Make-Up
         Tx_CB05_5 : Bool;   // Command 5 (LO): Emergency Setpoint On
         Tx_CB05_6 : Bool;   // Command 5 (LO): Emergency Setpoint Off
         Tx_CB05_7 : Bool;   // Command 5 (LO): Meas Drive On
         Tx_CW06 : Int;   // Command ID 2: Absolute Setpoint ID (250 Hex / 592 Dec)
         Tx_CD08_SP : Real;   // Absolute Setpoint [kg/h]
         Tx_CW12 : Int;   // Command ID 3: Command 6 + 7 (160 Hex / 352 Dec)
         Tx_CB14_0 : Bool;   // Command 6 (HI): Bin controller Autom.
         Tx_CB14_1 : Bool;   // Command 6 (HI): Bin controller Manual
         Tx_CB14_2 : Bool;   // Command 6 (HI): Bin controller Man. Start
         Tx_CB14_3 : Bool;   // Command 6 (HI): Bin controller Man Stop
         Tx_CB14_4 : Bool;   // Command 6 (HI): Optimization Bin Controller
         Tx_CB14_5 : Bool;   // Command 6 (HI): Print check Meas. Result
         Tx_CB14_6 : Bool;   // Command 6 (HI): Dead Time preassign
         Tx_CB14_7 : Bool;   // Command 6 (HI): Dead Time initialize
         Tx_CB15_0_StrTara : Bool;   // Command 6 (LO): Start internal check for tara
         Tx_CB15_1_StrRange : Bool;   // Command 6 (LO): Start internal check for range
         Tx_CB15_2_Acquire : Bool;   // Command 6 (LO): Acquire check result
         Tx_CB15_3_Cancel : Bool;   // Command 6 (LO): Cancel check measurement
         Tx_CB15_4 : Bool;   // Command 6 (LO): Release check system
         Tx_CB15_5 : Bool;   // Command 6 (LO): Acquire ext. corr. factor for tare
         Tx_CB15_6 : Bool;   // Command 6 (LO): Acquire ext. corr. factor for range
         Tx_CB15_7 : Bool;   // Command 6 (LO): Start external check
         Tx_CB16_0 : Bool;   // Command 7 (HI): Linearization P4
         Tx_CB16_1 : Bool;   // Command 7 (HI): Volmetric
         Tx_CB16_2 : Bool;   // Command 7 (HI): Optimize controller
         Tx_CB16_3 : Bool;   // Command 7 (HI): Calibration Acquire
         Tx_CB16_4 : Bool;   // Command 7 (HI): Calibration Abort
         Tx_CB16_5 : Bool;   // Command 7 (HI): Time Acquire
         Tx_CB16_6 : Bool;   // Command 7 (HI): Bin: Tare
         Tx_CB16_7 : Bool;   // Command 7 (HI): Bin: Weight Check
         Tx_CB17_0 : Bool;   // Command 7 (LO): Tare
         Tx_CB17_1 : Bool;   // Command 7 (LO): Zero Set
         Tx_CB17_2 : Bool;   // Command 7 (LO): Weight Check
         Tx_CB17_3 : Bool;   // Command 7 (LO): Pulses/Revolution
         Tx_CB17_4 : Bool;   // Command 7 (LO): DAE Adjustment
         Tx_CB17_5 : Bool;   // Command 7 (LO): Liniarization P1
         Tx_CB17_6 : Bool;   // Command 7 (LO): Liniarization P2
         Tx_CB17_7 : Bool;   // Command 7 (LO): Liniarization P3
         Tx_CW18 : Int;   // Command ID 4: Command 10 + 11 (1A0 Hex / 416 Dec)
         Tx_CB20_0 : Bool;   // Command 10 (HI): Reset Sum of Component 9
         Tx_CB20_1 : Bool;   // Command 10 (HI): Reset Sum of Component 10
         Tx_CB20_2 : Bool;   // Command 10 (HI): Reset Sum of Batches
         Tx_CB20_3_FillStopped : Bool;   // Command 10 (HI): Filling Stopped
         Tx_CB20_4 : Bool;   // Command 10 (HI): Start (static)
         Tx_CB20_5 : Bool;   // Command 10 (HI):
         Tx_CB20_6 : Bool;   // Command 10 (HI): Activate 2nd Batch Unit
         Tx_CB20_7 : Bool;   // Command 10 (HI): De-activate 2nd Batch Unit
         Tx_CB21_0 : Bool;   // Command 10 (LO): Reset Sum of Component 1
         Tx_CB21_1 : Bool;   // Command 10 (LO): Reset Sum of Component 2
         Tx_CB21_2 : Bool;   // Command 10 (LO): Reset Sum of Component 3
         Tx_CB21_3 : Bool;   // Command 10 (LO): Reset Sum of Component 4
         Tx_CB21_4 : Bool;   // Command 10 (LO): Reset Sum of Component 5
         Tx_CB21_5 : Bool;   // Command 10 (LO): Reset Sum of Component 6
         Tx_CB21_6 : Bool;   // Command 10 (LO): Reset Sum of Component 7
         Tx_CB21_7 : Bool;   // Command 10 (LO): Reset Sum of Component 8
         Tx_CB22_0 : Bool;   // Command 11 (HI): Feeder 1 Active
         Tx_CB22_1 : Bool;   // Command 11 (HI): Feeder 1 Not Active
         Tx_CB22_2 : Bool;   // Command 11 (HI): Feeder 1 Active
         Tx_CB22_3 : Bool;   // Command 11 (HI): Feeder 1 Not Active
         Tx_CB22_4 : Bool;   // Command 11 (HI): Set Norminal Feed Rate
         Tx_CB22_5 : Bool;   // Command 11 (HI): Copy feed index block
         Tx_CB22_6 : Bool;   // Command 11 (HI):
         Tx_CB22_7 : Bool;   // Command 11 (HI):
         Tx_CB23 : Byte;   // Command 11 (LO): Component Number (1 Byte)
         Tx_CW24 : Int;   // Status ID 1: Totalizer 1 [kg] (752 Hex / 1874 Dec)
         Tx_CW26 : Int;   // Status ID 2: Bin Weigher Fill Weight [kg] (762 Hex / 1890 Dec)
         Tx_CW28 : Int;   // Status ID 3: Status 0 + 1 (2D0 Hex / 720 Dec)
         Tx_CW30 : Int;   // Status ID 4: Status 8 + 9 (350 Hex / 848 Dec)
         Tx_CW32 : Int;   // Status ID 5: Priority Event (610 Hex / 1552 Dec)
         Tx_CW34 : Int;   // Status ID 6: Varialbe ID from faceplate range 1872-2158 (dec)
         Tx_CW36 : Int;   // Status ID 7: Status 4 + 5 (310 Hex / 784 Dec)
         Tx_CW38 : Int;   // Status ID 8: Check Result F/Z (7EA Hex / 2026 Dec)
         Tx_CW40 : Int;   // Status ID 9: Actual Setpoint [kg/h] (766 Hex / 1894 Dec)
         Tx_CW42 : Int;   // Status ID 10: Deviation (770 Hex / 1904 Dec)
         Tx_CW44 : Int;   // Status ID 11: Not Used (0 Hex / 0 Dec)
         Tx_CW46 : Int;   // Status ID 12: Not Used (0 Hex / 0 Dec)
      END_STRUCT;
      INTECONT : Struct
         Tx_CW00 : Int;   // Command ID 1: Command 4+5 (140 Hex / 320 Dec)
         Tx_CB02_0 : Bool;   // Command 4 (HI): Volm. Synchronous
         Tx_CB02_1 : Bool;   // Command 4 (HI): Moisture Corr. On
         Tx_CB02_2 : Bool;   // Command 4 (HI): Moisture Corr. Off
         Tx_CB02_3 : Bool;   // Command 4 (HI): Meas. Drive Off
         Tx_CB02_4 : Bool;   // Command 4 (HI): Gate Feedback
         Tx_CB02_5 : Bool;   // Command 4 (HI): Open Gate Manual
         Tx_CB02_6 : Bool;   // Command 4 (HI): Stop Gate Manual
         Tx_CB02_7 : Bool;   // Command 4 (HI): Close Gate Manual
         Tx_CB03_0_StrScale : Bool;   // Command 4 (LO): Start Scale
         Tx_CB03_1_StpScale : Bool;   // Command 4 (LO): Stop Scale
         Tx_CB03_2_ClearEvent : Bool;   // Command 4 (LO): Clear Events (RESET)
         Tx_CB03_3_Release : Bool;   // Command 4 (LO): Release
         Tx_CB03_4_SelVol : Bool;   // Command 4 (LO): Select Volumetric Mode
         Tx_CB03_5_SelGrav : Bool;   // Command 4 (LO): Select Gravimetric Mode
         Tx_CB03_6_ResTot : Bool;   // Command 4 (LO): Reset Totalizer 1
         Tx_CB03_7 : Bool;   // Command 4 (LO): Reset Totalizer 2
         Tx_CB04_0 : Bool;   // Command 5 (HI): Filling Start
         Tx_CB04_1 : Bool;   // Command 5 (HI): Filling Stop
         Tx_CB04_2 : Bool;   // Command 5 (HI): Emptying Start
         Tx_CB04_3 : Bool;   // Command 5 (HI): Emptying Stop
         Tx_CB04_4 : Bool;   // Command 5 (HI): Init .Hopper Controller
         Tx_CB04_5 : Bool;   // Command 5 (HI): Activate Fill Unit
         Tx_CB04_6 : Bool;   // Command 5 (HI): Activate Prefeeder
         Tx_CB04_7 : Bool;   // Command 5 (HI): Stop Prefeeder
         Tx_CB05_0 : Bool;   // Command 5 (LO): Select Batch
         Tx_CB05_1 : Bool;   // Command 5 (LO): Deselect Batch
         Tx_CB05_2 : Bool;   // Command 5 (LO): Abort Batch
         Tx_CB05_3 : Bool;   // Command 5 (LO): Next Batch + Clearance
         Tx_CB05_4 : Bool;   // Command 5 (LO): Make-Up
         Tx_CB05_5 : Bool;   // Command 5 (LO): Emergency Setpoint On
         Tx_CB05_6 : Bool;   // Command 5 (LO): Emergency Setpoint Off
         Tx_CB05_7 : Bool;   // Command 5 (LO): Meas Drive On
         Tx_CW06 : Int;   // Command ID 2: Absolute Setpoint ID (250 Hex / 592 Dec)
         Tx_CD08_SP : Real;   // Absolute Setpoint [kg/h]
         Tx_CW12 : Int;   // Command ID 3: Command 6 + 7 (160 Hex / 352 Dec)
         Tx_CB14_0 : Bool;   // Command 6 (HI): Bin controller Autom.
         Tx_CB14_1 : Bool;   // Command 6 (HI): Bin controller Manual
         Tx_CB14_2 : Bool;   // Command 6 (HI): Bin controller Man. Start
         Tx_CB14_3 : Bool;   // Command 6 (HI): Bin controller Man Stop
         Tx_CB14_4 : Bool;   // Command 6 (HI): Optimization Bin Controller
         Tx_CB14_5 : Bool;   // Command 6 (HI): Print check Meas. Result
         Tx_CB14_6 : Bool;   // Command 6 (HI): Dead Time preassign
         Tx_CB14_7 : Bool;   // Command 6 (HI): Dead Time initialize
         Tx_CB15_0_StrTara : Bool;   // Command 6 (LO): Start internal check for tara
         Tx_CB15_1_StrRange : Bool;   // Command 6 (LO): Start internal check for range
         Tx_CB15_2_Acquire : Bool;   // Command 6 (LO): Acquire check result
         Tx_CB15_3_Cancel : Bool;   // Command 6 (LO): Cancel check measurement
         Tx_CB15_4 : Bool;   // Command 6 (LO): Release check system
         Tx_CB15_5 : Bool;   // Command 6 (LO): Acquire ext. corr. factor for tare
         Tx_CB15_6 : Bool;   // Command 6 (LO): Acquire ext. corr. factor for range
         Tx_CB15_7 : Bool;   // Command 6 (LO): Start external check
         Tx_CB16_0 : Bool;   // Command 7 (HI): Linearization P4
         Tx_CB16_1 : Bool;   // Command 7 (HI): Volmetric
         Tx_CB16_2 : Bool;   // Command 7 (HI): Optimize controller
         Tx_CB16_3 : Bool;   // Command 7 (HI): Calibration Acquire
         Tx_CB16_4 : Bool;   // Command 7 (HI): Calibration Abort
         Tx_CB16_5 : Bool;   // Command 7 (HI): Time Acquire
         Tx_CB16_6 : Bool;   // Command 7 (HI): Bin: Tare
         Tx_CB16_7 : Bool;   // Command 7 (HI): Bin: Weight Check
         Tx_CB17_0 : Bool;   // Command 7 (LO): Tare
         Tx_CB17_1 : Bool;   // Command 7 (LO): Zero Set
         Tx_CB17_2 : Bool;   // Command 7 (LO): Weight Check
         Tx_CB17_3 : Bool;   // Command 7 (LO): Pulses/Revolution
         Tx_CB17_4 : Bool;   // Command 7 (LO): DAE Adjustment
         Tx_CB17_5 : Bool;   // Command 7 (LO): Liniarization P1
         Tx_CB17_6 : Bool;   // Command 7 (LO): Liniarization P2
         Tx_CB17_7 : Bool;   // Command 7 (LO): Liniarization P3
         Tx_CW18 : Int;   // Status ID 1: Totalizer 1 [kg] (752 Hex / 1874 Dec)
         Tx_CW20 : Int;   // Status ID 2: Bin Weigher Fill Weight [kg] (762 Hex / 1890 Dec)
         Tx_CW22 : Int;   // Status ID 3: Status 0 + 1 (2D0 Hex / 720 Dec)
         Tx_CW24 : Int;   // Status ID 4: Status 8 + 9 (350 Hex / 848 Dec)
         Tx_CW26 : Int;   // Status ID 5: Priority Event (610 Hex / 1552 Dec)
         Tx_CW28 : Int;   // Status ID 6: Variable ID from faceplate range 1872-2158 (dec)
      END_STRUCT;
      AOn : Bool;   // Always On
      AOff : Bool;   // Always Off
      DummyBool : Bool;
      Temp_CON : Bool;
      TYPE_INTECONT : Bool;
      TYPE_DISOCONT : Bool;
      BusFault : Bool;   // Bus failure
      StatPointer_Old : Int;
      StatusBuilder : Int;
      TempReal : Real;
      TempDINT : DInt;
      TempInt : Int;
      TempDword : DWord;
      TempWord : Word;
      MaskWord : Word;
      TempByte : Byte;
      BlkMov_Status : Int;
      PackageLength : Int;
      Schenck_offset : Int;
      ScaleTypeNo : Int;   // 1=VDB, 2=VBW, 4=VDD, 5=VDM, 9=VMD
      Addr_InstanceDB : DWord;
      DB_Pointer : ANY;
      IO_Pointer : ANY;
      DelayedCMD : Bool;
      Status_Add : Int;
   END_VAR
   VAR_TEMP   // added for the SCL form of the ladder/FBD networks
      _w1 : Bool;
      _w2 : Bool;
      _w3 : Bool;
      _w4 : Bool;
      _w5 : Bool;
      _w6 : Bool;
   END_VAR
BEGIN

REGION Network 1: Always On
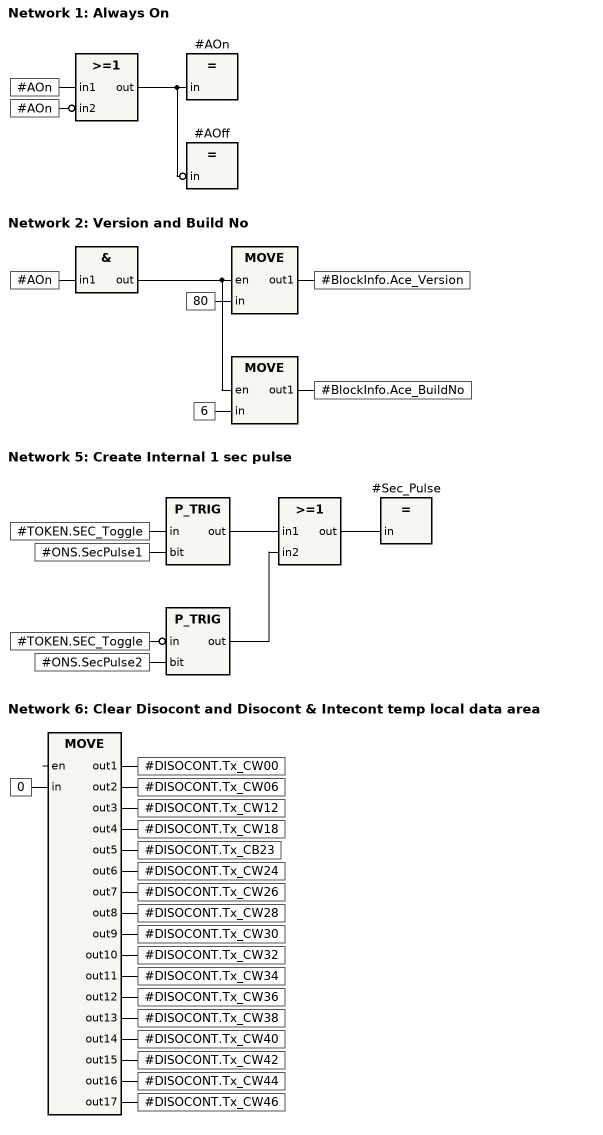
   #AOn := #AOn OR NOT #AOn;
   #AOff := NOT #AOn;
END_REGION

REGION Network 2: Version and Build No
   IF #AOn THEN
       #BlockInfo.Ace_Version := 80;
       #BlockInfo.Ace_BuildNo := 6;
   END_IF;
END_REGION

REGION Network 3 (STL): Instance DB Number to Faceplate
         L     DINO;
         T     #BlockInfo.DB_Number;
END_REGION

REGION Network 4 (SCL): Transfer Interlock OK to Stat
   #OUT.INTL_OK_STAT := PEEK_BOOL(area := 16#84, dbNumber := #BlockInfo.DB_Number, byteOffset := 20, bitOffset := 0);
   #OUT.INTL_SEQ_STR_OK_STAT := PEEK_BOOL(area := 16#84, dbNumber := #BlockInfo.DB_Number, byteOffset := 22, bitOffset := 0);
   #OUT.INTL_SEQ_STP_OK_STAT := PEEK_BOOL(area := 16#84, dbNumber := #BlockInfo.DB_Number, byteOffset := 24, bitOffset := 0);
END_REGION

REGION Network 5: Create Internal 1 sec pulse
   #_w1 := #TOKEN.SEC_Toggle AND NOT #ONS.SecPulse1;   // rising edge
   #ONS.SecPulse1 := #TOKEN.SEC_Toggle;
   #_w2 := NOT #TOKEN.SEC_Toggle AND NOT #ONS.SecPulse2;   // rising edge
   #ONS.SecPulse2 := NOT #TOKEN.SEC_Toggle;
   #Sec_Pulse := #_w1 OR #_w2;
END_REGION

REGION Network 6: Clear Disocont and Disocont & Intecont temp local data area
   #DISOCONT.Tx_CW00 := 0;
   #DISOCONT.Tx_CW06 := 0;
   #DISOCONT.Tx_CW12 := 0;
   #DISOCONT.Tx_CW18 := 0;
   #DISOCONT.Tx_CB23 := 0;
   #DISOCONT.Tx_CW24 := 0;
   #DISOCONT.Tx_CW26 := 0;
   #DISOCONT.Tx_CW28 := 0;
   #DISOCONT.Tx_CW30 := 0;
   #DISOCONT.Tx_CW32 := 0;
   #DISOCONT.Tx_CW34 := 0;
   #DISOCONT.Tx_CW36 := 0;
   #DISOCONT.Tx_CW38 := 0;
   #DISOCONT.Tx_CW40 := 0;
   #DISOCONT.Tx_CW42 := 0;
   #DISOCONT.Tx_CW44 := 0;
   #DISOCONT.Tx_CW46 := 0;
END_REGION

REGION Network 7: DISOCONT - Reset - Byte 2 & 3
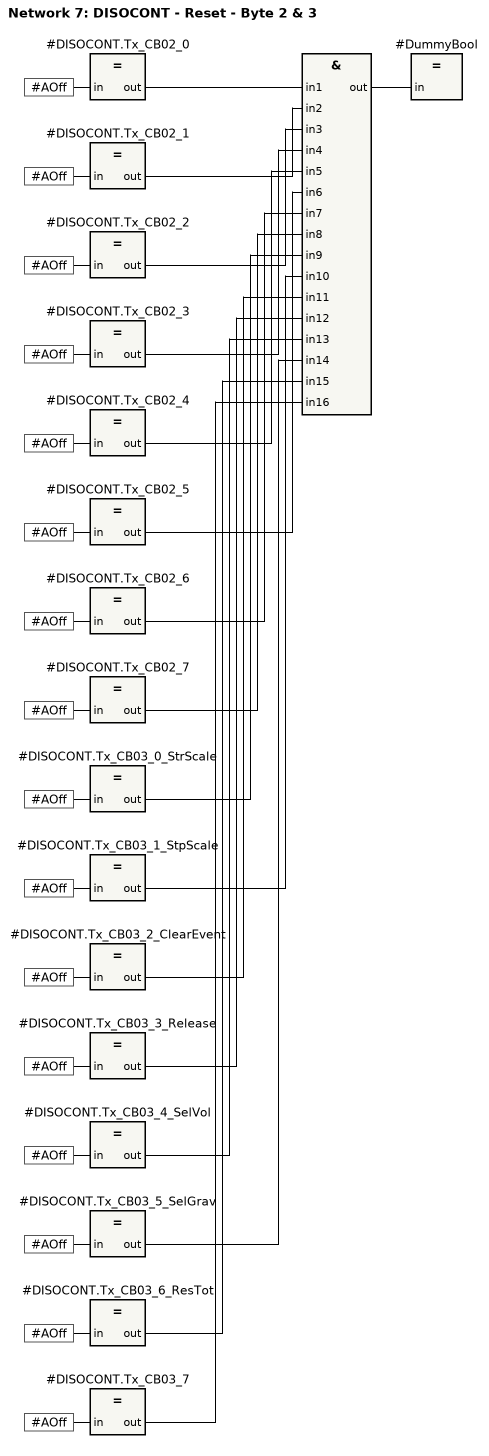
   #DISOCONT.Tx_CB02_0 := #AOff;
   #DISOCONT.Tx_CB02_1 := #AOff;
   #DISOCONT.Tx_CB02_2 := #AOff;
   #DISOCONT.Tx_CB02_3 := #AOff;
   #DISOCONT.Tx_CB02_4 := #AOff;
   #DISOCONT.Tx_CB02_5 := #AOff;
   #DISOCONT.Tx_CB02_6 := #AOff;
   #DISOCONT.Tx_CB02_7 := #AOff;
   #DISOCONT.Tx_CB03_0_StrScale := #AOff;
   #DISOCONT.Tx_CB03_1_StpScale := #AOff;
   #DISOCONT.Tx_CB03_2_ClearEvent := #AOff;
   #DISOCONT.Tx_CB03_3_Release := #AOff;
   #DISOCONT.Tx_CB03_4_SelVol := #AOff;
   #DISOCONT.Tx_CB03_5_SelGrav := #AOff;
   #DISOCONT.Tx_CB03_6_ResTot := #AOff;
   #DISOCONT.Tx_CB03_7 := #AOff;
   #DummyBool := #AOff AND #AOff AND #AOff AND #AOff AND #AOff AND #AOff AND #AOff AND #AOff AND #AOff AND #AOff AND #AOff AND #AOff AND #AOff AND #AOff AND #AOff AND #AOff;
END_REGION

REGION Network 8: DISOCONT - Reset - Byte 4 & 5
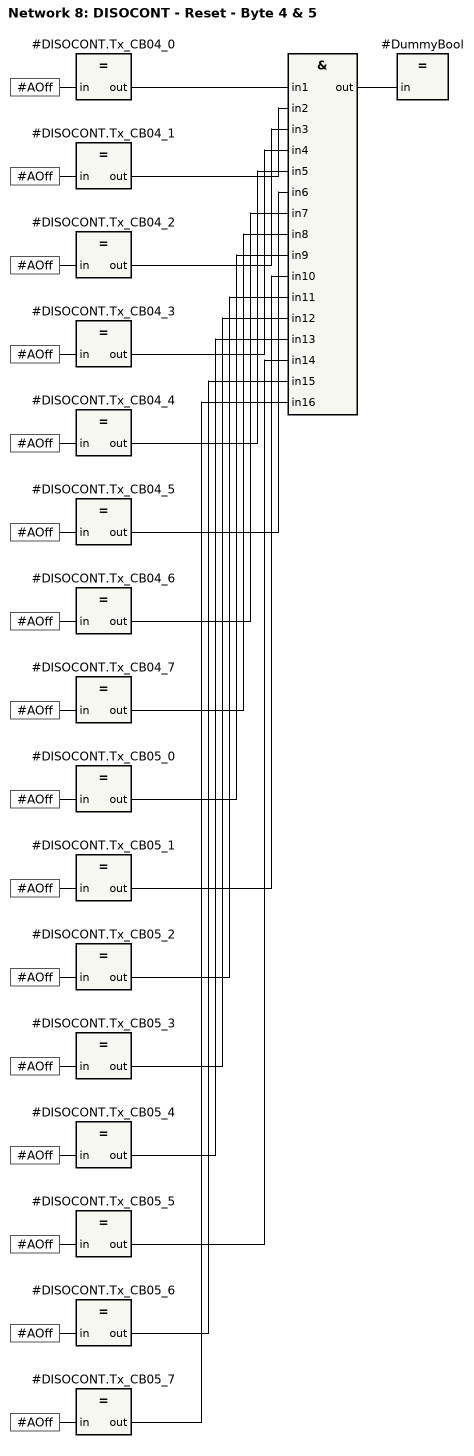
   #DISOCONT.Tx_CB04_0 := #AOff;
   #DISOCONT.Tx_CB04_1 := #AOff;
   #DISOCONT.Tx_CB04_2 := #AOff;
   #DISOCONT.Tx_CB04_3 := #AOff;
   #DISOCONT.Tx_CB04_4 := #AOff;
   #DISOCONT.Tx_CB04_5 := #AOff;
   #DISOCONT.Tx_CB04_6 := #AOff;
   #DISOCONT.Tx_CB04_7 := #AOff;
   #DISOCONT.Tx_CB05_0 := #AOff;
   #DISOCONT.Tx_CB05_1 := #AOff;
   #DISOCONT.Tx_CB05_2 := #AOff;
   #DISOCONT.Tx_CB05_3 := #AOff;
   #DISOCONT.Tx_CB05_4 := #AOff;
   #DISOCONT.Tx_CB05_5 := #AOff;
   #DISOCONT.Tx_CB05_6 := #AOff;
   #DISOCONT.Tx_CB05_7 := #AOff;
   #DummyBool := #AOff AND #AOff AND #AOff AND #AOff AND #AOff AND #AOff AND #AOff AND #AOff AND #AOff AND #AOff AND #AOff AND #AOff AND #AOff AND #AOff AND #AOff AND #AOff;
END_REGION

REGION Network 9
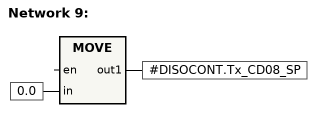
   #DISOCONT.Tx_CD08_SP := 0.0;
END_REGION

REGION Network 10: DISOCONT - Reset - Byte 14 & 15
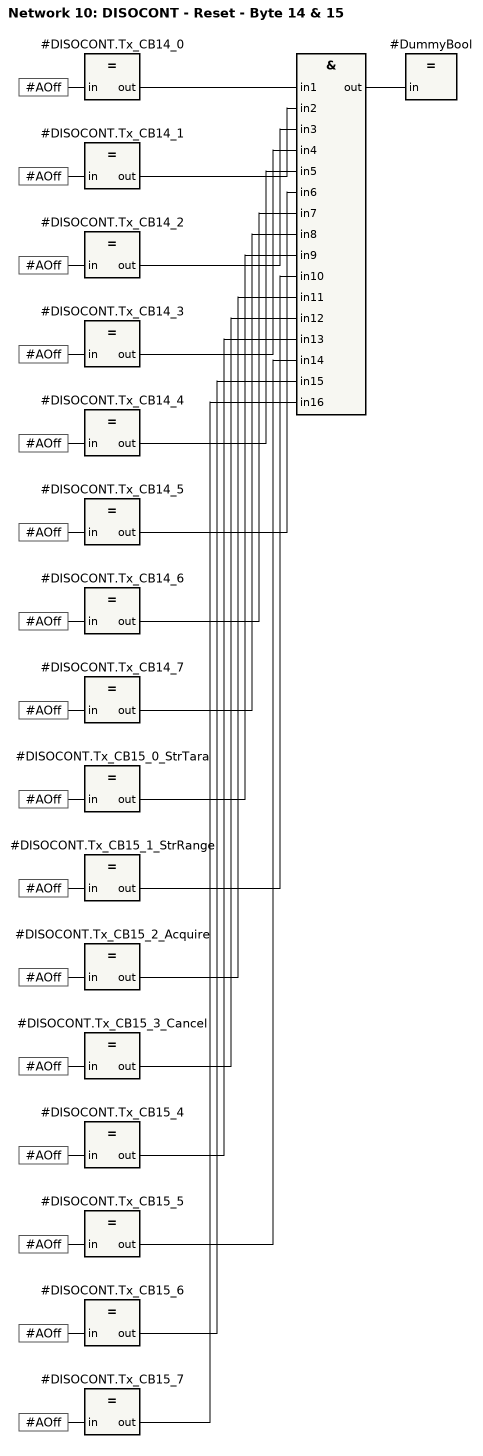
   #DISOCONT.Tx_CB14_0 := #AOff;
   #DISOCONT.Tx_CB14_1 := #AOff;
   #DISOCONT.Tx_CB14_2 := #AOff;
   #DISOCONT.Tx_CB14_3 := #AOff;
   #DISOCONT.Tx_CB14_4 := #AOff;
   #DISOCONT.Tx_CB14_5 := #AOff;
   #DISOCONT.Tx_CB14_6 := #AOff;
   #DISOCONT.Tx_CB14_7 := #AOff;
   #DISOCONT.Tx_CB15_0_StrTara := #AOff;
   #DISOCONT.Tx_CB15_1_StrRange := #AOff;
   #DISOCONT.Tx_CB15_2_Acquire := #AOff;
   #DISOCONT.Tx_CB15_3_Cancel := #AOff;
   #DISOCONT.Tx_CB15_4 := #AOff;
   #DISOCONT.Tx_CB15_5 := #AOff;
   #DISOCONT.Tx_CB15_6 := #AOff;
   #DISOCONT.Tx_CB15_7 := #AOff;
   #DummyBool := #AOff AND #AOff AND #AOff AND #AOff AND #AOff AND #AOff AND #AOff AND #AOff AND #AOff AND #AOff AND #AOff AND #AOff AND #AOff AND #AOff AND #AOff AND #AOff;
END_REGION

REGION Network 11: DISOCONT - Reset - Byte 16 & 17
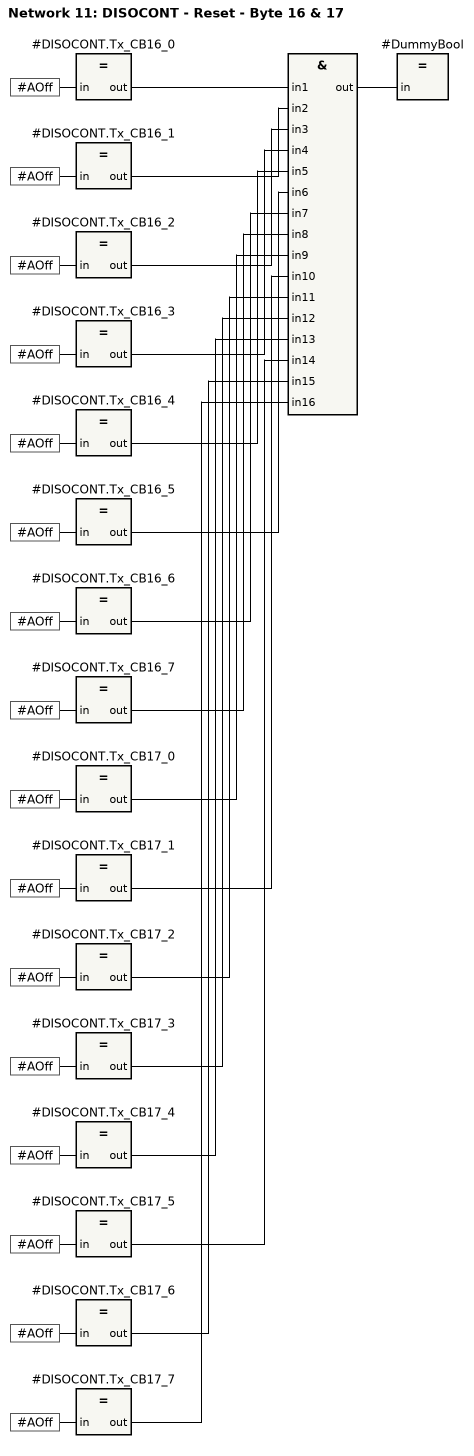
   #DISOCONT.Tx_CB16_0 := #AOff;
   #DISOCONT.Tx_CB16_1 := #AOff;
   #DISOCONT.Tx_CB16_2 := #AOff;
   #DISOCONT.Tx_CB16_3 := #AOff;
   #DISOCONT.Tx_CB16_4 := #AOff;
   #DISOCONT.Tx_CB16_5 := #AOff;
   #DISOCONT.Tx_CB16_6 := #AOff;
   #DISOCONT.Tx_CB16_7 := #AOff;
   #DISOCONT.Tx_CB17_0 := #AOff;
   #DISOCONT.Tx_CB17_1 := #AOff;
   #DISOCONT.Tx_CB17_2 := #AOff;
   #DISOCONT.Tx_CB17_3 := #AOff;
   #DISOCONT.Tx_CB17_4 := #AOff;
   #DISOCONT.Tx_CB17_5 := #AOff;
   #DISOCONT.Tx_CB17_6 := #AOff;
   #DISOCONT.Tx_CB17_7 := #AOff;
   #DummyBool := #AOff AND #AOff AND #AOff AND #AOff AND #AOff AND #AOff AND #AOff AND #AOff AND #AOff AND #AOff AND #AOff AND #AOff AND #AOff AND #AOff AND #AOff AND #AOff;
END_REGION

REGION Network 12: DISOCONT - Reset - Byte 20 & 21
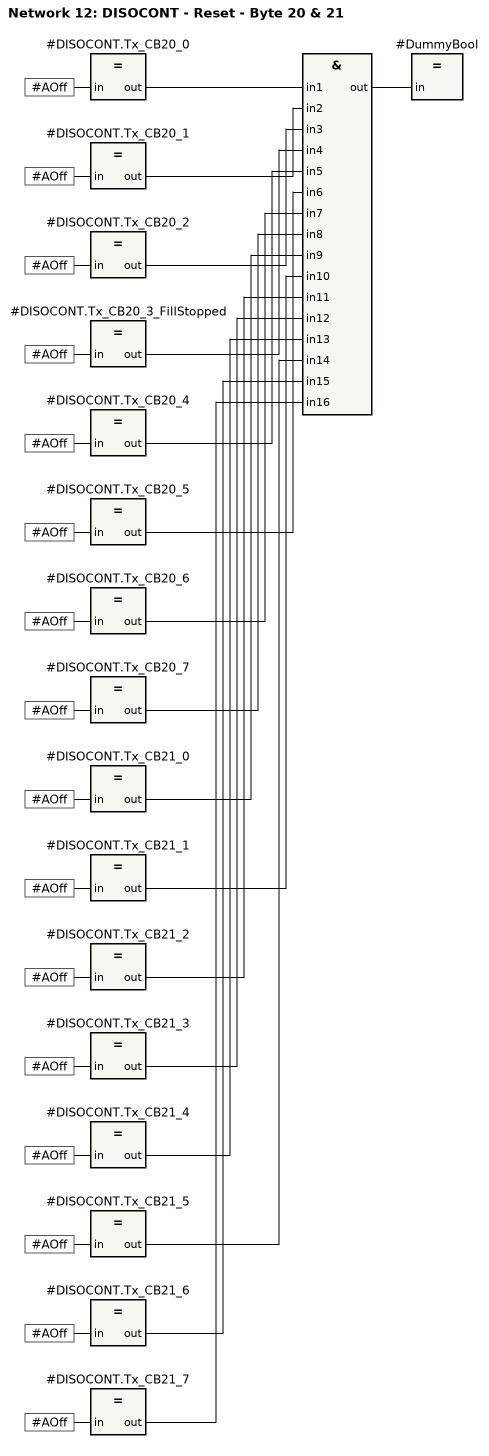
   #DISOCONT.Tx_CB20_0 := #AOff;
   #DISOCONT.Tx_CB20_1 := #AOff;
   #DISOCONT.Tx_CB20_2 := #AOff;
   #DISOCONT.Tx_CB20_3_FillStopped := #AOff;
   #DISOCONT.Tx_CB20_4 := #AOff;
   #DISOCONT.Tx_CB20_5 := #AOff;
   #DISOCONT.Tx_CB20_6 := #AOff;
   #DISOCONT.Tx_CB20_7 := #AOff;
   #DISOCONT.Tx_CB21_0 := #AOff;
   #DISOCONT.Tx_CB21_1 := #AOff;
   #DISOCONT.Tx_CB21_2 := #AOff;
   #DISOCONT.Tx_CB21_3 := #AOff;
   #DISOCONT.Tx_CB21_4 := #AOff;
   #DISOCONT.Tx_CB21_5 := #AOff;
   #DISOCONT.Tx_CB21_6 := #AOff;
   #DISOCONT.Tx_CB21_7 := #AOff;
   #DummyBool := #AOff AND #AOff AND #AOff AND #AOff AND #AOff AND #AOff AND #AOff AND #AOff AND #AOff AND #AOff AND #AOff AND #AOff AND #AOff AND #AOff AND #AOff AND #AOff;
END_REGION

REGION Network 13: DISOCONT - Reset - Byte 22
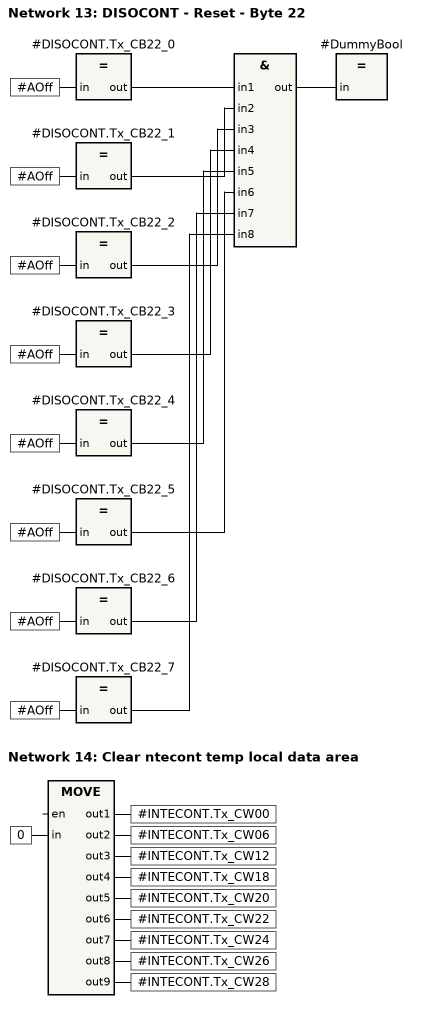
   #DISOCONT.Tx_CB22_0 := #AOff;
   #DISOCONT.Tx_CB22_1 := #AOff;
   #DISOCONT.Tx_CB22_2 := #AOff;
   #DISOCONT.Tx_CB22_3 := #AOff;
   #DISOCONT.Tx_CB22_4 := #AOff;
   #DISOCONT.Tx_CB22_5 := #AOff;
   #DISOCONT.Tx_CB22_6 := #AOff;
   #DISOCONT.Tx_CB22_7 := #AOff;
   #DummyBool := #AOff AND #AOff AND #AOff AND #AOff AND #AOff AND #AOff AND #AOff AND #AOff;
END_REGION

REGION Network 14: Clear ntecont temp local data area
   #INTECONT.Tx_CW00 := 0;
   #INTECONT.Tx_CW06 := 0;
   #INTECONT.Tx_CW12 := 0;
   #INTECONT.Tx_CW18 := 0;
   #INTECONT.Tx_CW20 := 0;
   #INTECONT.Tx_CW22 := 0;
   #INTECONT.Tx_CW24 := 0;
   #INTECONT.Tx_CW26 := 0;
   #INTECONT.Tx_CW28 := 0;
END_REGION

REGION Network 15: INTECONT - Reset - Byte 2 & 3
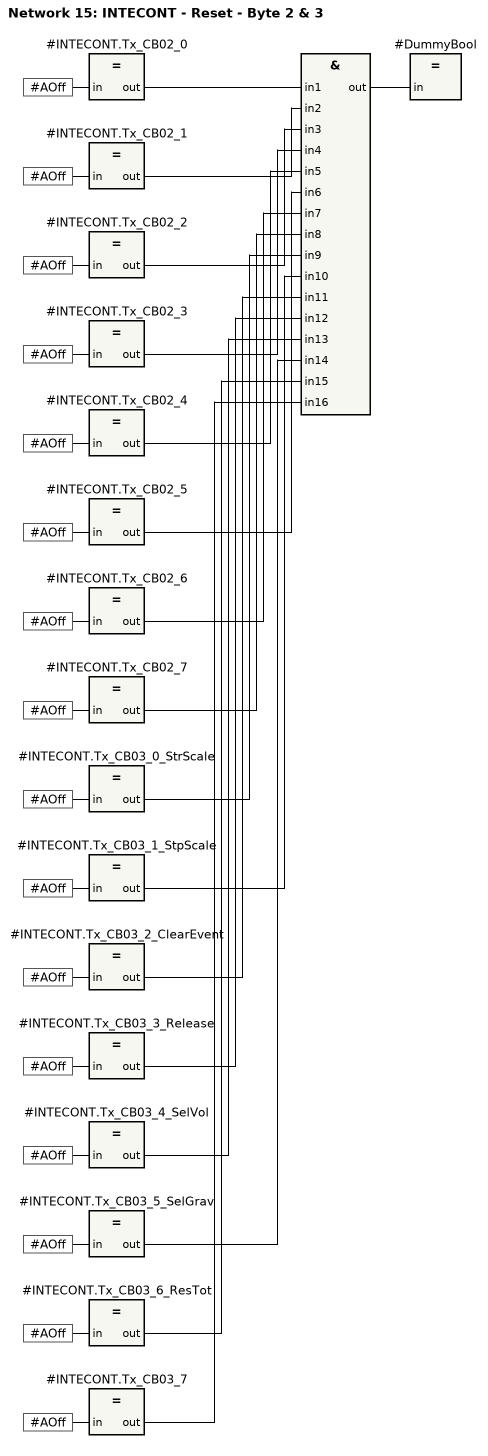
   #INTECONT.Tx_CB02_0 := #AOff;
   #INTECONT.Tx_CB02_1 := #AOff;
   #INTECONT.Tx_CB02_2 := #AOff;
   #INTECONT.Tx_CB02_3 := #AOff;
   #INTECONT.Tx_CB02_4 := #AOff;
   #INTECONT.Tx_CB02_5 := #AOff;
   #INTECONT.Tx_CB02_6 := #AOff;
   #INTECONT.Tx_CB02_7 := #AOff;
   #INTECONT.Tx_CB03_0_StrScale := #AOff;
   #INTECONT.Tx_CB03_1_StpScale := #AOff;
   #INTECONT.Tx_CB03_2_ClearEvent := #AOff;
   #INTECONT.Tx_CB03_3_Release := #AOff;
   #INTECONT.Tx_CB03_4_SelVol := #AOff;
   #INTECONT.Tx_CB03_5_SelGrav := #AOff;
   #INTECONT.Tx_CB03_6_ResTot := #AOff;
   #INTECONT.Tx_CB03_7 := #AOff;
   #DummyBool := #AOff AND #AOff AND #AOff AND #AOff AND #AOff AND #AOff AND #AOff AND #AOff AND #AOff AND #AOff AND #AOff AND #AOff AND #AOff AND #AOff AND #AOff AND #AOff;
END_REGION

REGION Network 16: INTECONT - Reset - Byte 4 & 5
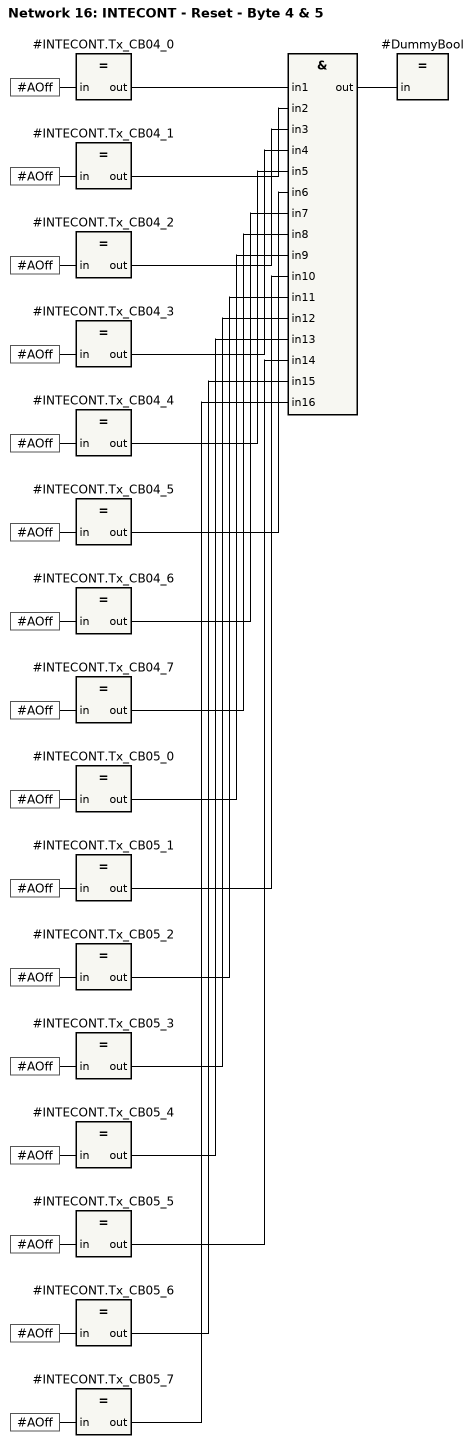
   #INTECONT.Tx_CB04_0 := #AOff;
   #INTECONT.Tx_CB04_1 := #AOff;
   #INTECONT.Tx_CB04_2 := #AOff;
   #INTECONT.Tx_CB04_3 := #AOff;
   #INTECONT.Tx_CB04_4 := #AOff;
   #INTECONT.Tx_CB04_5 := #AOff;
   #INTECONT.Tx_CB04_6 := #AOff;
   #INTECONT.Tx_CB04_7 := #AOff;
   #INTECONT.Tx_CB05_0 := #AOff;
   #INTECONT.Tx_CB05_1 := #AOff;
   #INTECONT.Tx_CB05_2 := #AOff;
   #INTECONT.Tx_CB05_3 := #AOff;
   #INTECONT.Tx_CB05_4 := #AOff;
   #INTECONT.Tx_CB05_5 := #AOff;
   #INTECONT.Tx_CB05_6 := #AOff;
   #INTECONT.Tx_CB05_7 := #AOff;
   #DummyBool := #AOff AND #AOff AND #AOff AND #AOff AND #AOff AND #AOff AND #AOff AND #AOff AND #AOff AND #AOff AND #AOff AND #AOff AND #AOff AND #AOff AND #AOff AND #AOff;
END_REGION

REGION Network 17
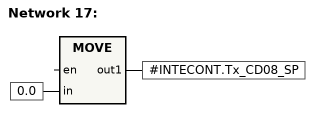
   #INTECONT.Tx_CD08_SP := 0.0;
END_REGION

REGION Network 18: INTECONT - Reset - Byte 14 & 15
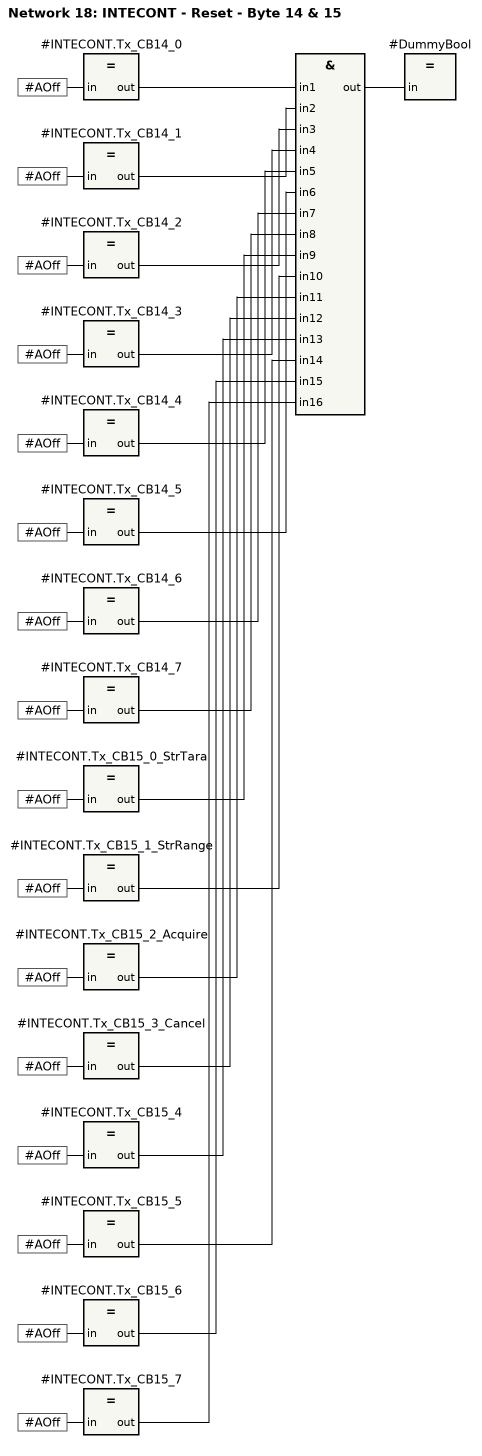
   #INTECONT.Tx_CB14_0 := #AOff;
   #INTECONT.Tx_CB14_1 := #AOff;
   #INTECONT.Tx_CB14_2 := #AOff;
   #INTECONT.Tx_CB14_3 := #AOff;
   #INTECONT.Tx_CB14_4 := #AOff;
   #INTECONT.Tx_CB14_5 := #AOff;
   #INTECONT.Tx_CB14_6 := #AOff;
   #INTECONT.Tx_CB14_7 := #AOff;
   #INTECONT.Tx_CB15_0_StrTara := #AOff;
   #INTECONT.Tx_CB15_1_StrRange := #AOff;
   #INTECONT.Tx_CB15_2_Acquire := #AOff;
   #INTECONT.Tx_CB15_3_Cancel := #AOff;
   #INTECONT.Tx_CB15_4 := #AOff;
   #INTECONT.Tx_CB15_5 := #AOff;
   #INTECONT.Tx_CB15_6 := #AOff;
   #INTECONT.Tx_CB15_7 := #AOff;
   #DummyBool := #AOff AND #AOff AND #AOff AND #AOff AND #AOff AND #AOff AND #AOff AND #AOff AND #AOff AND #AOff AND #AOff AND #AOff AND #AOff AND #AOff AND #AOff AND #AOff;
END_REGION

REGION Network 19: INTECONT - Reset - Byte 16 & 17
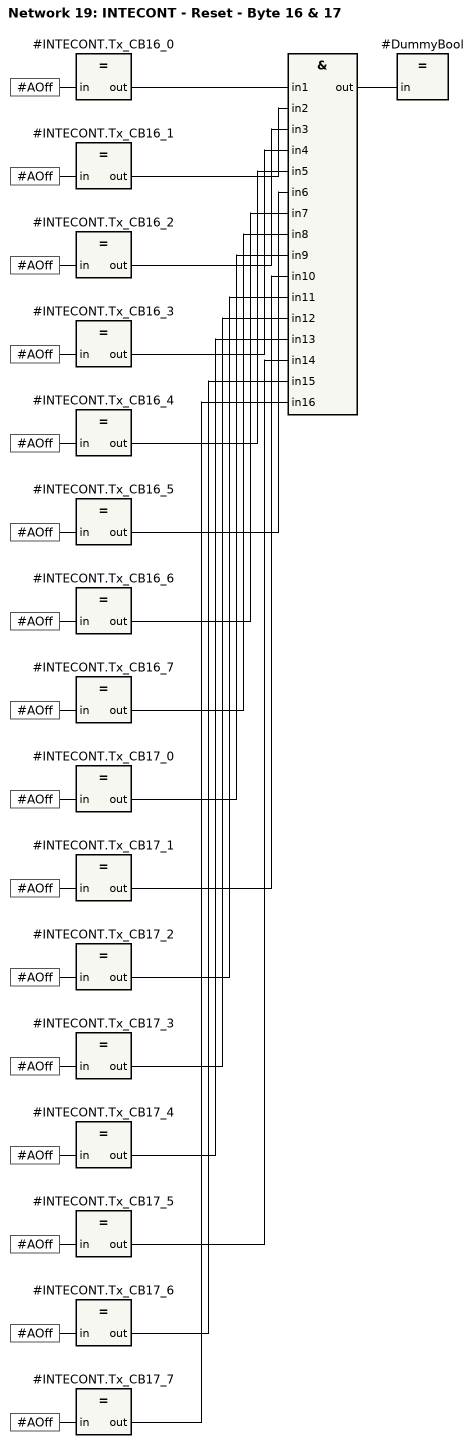
   #INTECONT.Tx_CB16_0 := #AOff;
   #INTECONT.Tx_CB16_1 := #AOff;
   #INTECONT.Tx_CB16_2 := #AOff;
   #INTECONT.Tx_CB16_3 := #AOff;
   #INTECONT.Tx_CB16_4 := #AOff;
   #INTECONT.Tx_CB16_5 := #AOff;
   #INTECONT.Tx_CB16_6 := #AOff;
   #INTECONT.Tx_CB16_7 := #AOff;
   #INTECONT.Tx_CB17_0 := #AOff;
   #INTECONT.Tx_CB17_1 := #AOff;
   #INTECONT.Tx_CB17_2 := #AOff;
   #INTECONT.Tx_CB17_3 := #AOff;
   #INTECONT.Tx_CB17_4 := #AOff;
   #INTECONT.Tx_CB17_5 := #AOff;
   #INTECONT.Tx_CB17_6 := #AOff;
   #INTECONT.Tx_CB17_7 := #AOff;
   #DummyBool := #AOff AND #AOff AND #AOff AND #AOff AND #AOff AND #AOff AND #AOff AND #AOff AND #AOff AND #AOff AND #AOff AND #AOff AND #AOff AND #AOff AND #AOff AND #AOff;
END_REGION

REGION Network 20: Set equipment Type: DISOCONT
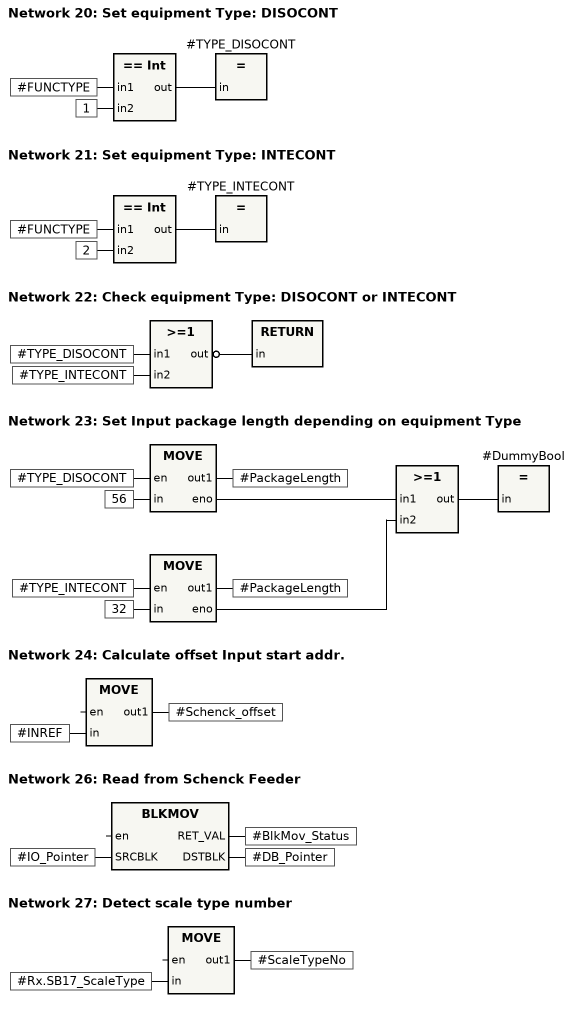
   #TYPE_DISOCONT := #FUNCTYPE = 1;
END_REGION

REGION Network 21: Set equipment Type: INTECONT
   #TYPE_INTECONT := #FUNCTYPE = 2;
END_REGION

REGION Network 22: Check equipment Type: DISOCONT or INTECONT
   IF NOT (#TYPE_DISOCONT OR #TYPE_INTECONT) THEN
       ENO := TRUE;
       RETURN;
   END_IF;
END_REGION

REGION Network 23: Set Input package length depending on equipment Type
   // ENO of a box is taken as its EN; it also drops when the box reports an error
   IF #TYPE_DISOCONT THEN #PackageLength := 56; END_IF;
   IF #TYPE_INTECONT THEN #PackageLength := 32; END_IF;
   #DummyBool := #TYPE_DISOCONT OR #TYPE_INTECONT;
END_REGION

REGION Network 24: Calculate offset Input start addr.
   // Hardware Address
   #Schenck_offset := #INREF;
END_REGION

REGION Network 25 (STL): Target Pointers Recieve input data
         LAR1;  // Make AR1 point to calling program stack
         L     16#10;  // ANY Syntax ID
         T     LB[AR1, P#0.0];  // ..Store Byte 0
         L     16#02;  // Data Type = Byte
         T     LB[AR1, P#1.0];  // ..Store Byte 1
         L     #PackageLength;  // Load Packed length
         T     LW[AR1, P#2.0];  // ..Store byte 2/3
         L     0;  // used with DB else "0"
         T     LW[AR1, P#4.0];  // ..Store byte 4/5
         L     #Schenck_offset;  // Source offset (Variable for Node's)
         SLD   3;  // with offset
         OD    16#8100_0000;  // Input Area (I/O) Code (S7)
         T     LD[AR1, P#6.0];  // ..Store byte 6/7/8/9

         LAR1;  // Load start point of cyclic data
         TAR1  #TempDword;  // Store in temp. point
         L     #TempDword;  // Load temp. point
         T     #Addr_InstanceDB;  // Store start point as DB address

         LAR1;  // Make AR1 point to calling program stack
         L     16#10;  // ANY Syntax ID
         T     LB[AR1, P#0.0];  // ..Store Byte 0
         L     16#02;  // Data Type = Byte
         T     LB[AR1, P#1.0];  // ..Store Byte 1
         L     #PackageLength;  // Load Packed length
         T     LW[AR1, P#2.0];  // ..Store Byte 2/3
         L     #BlockInfo.DB_Number;  // used with DB use No. else "0"
         T     LW[AR1, P#4.0];  // ..Store byte 4/5
         L     #Addr_InstanceDB;  // Load Instance DB Start address
         L     16#8500_0000;
         -D;
         L     16#8400_0000;
         +D;
         T     LD[AR1, P#6.0];  // ..Store byte 6/7/8/9
END_REGION

REGION Network 26: Read from Schenck Feeder
   #BlkMov_Status := BLKMOV(SRCBLK := #IO_Pointer, DSTBLK => #DB_Pointer);
END_REGION

REGION Network 27: Detect scale type number
   // Supported Scale types:
   // ScaleTypeNo = 1 = VDB = Weight Feeder
   // ScaleTypeNo = 2 = VBW = Belt Weight
   // ScaleTypeNo = 4 = VDD = Solid Flow Feeder
   // ScaleTypeNo = 5 = VDM = Solid Flow Meter
   // ScaleTypeNo = 9 = VMD = Mass Flow Feeder
   #ScaleTypeNo := #Rx.SB17_ScaleType;
END_REGION

REGION Network 28: Unknown Scale Type Error
   // On error rest of the block is skipped.
   // Build 004 - 24. July 2019 (EXTBOB): New type 39 added for Disocont Tersus (To be tested)
